LIN {X 0,Y 227.734,Z 309.956,A -85,B 0,C 180,E1 -22009.411,E2 -22009.411} C_VEL
LIN {X 0,Y 228.361,Z 312.963,A -85,B 0,C 180,E1 -22009.7,E2 -22009.7} C_VEL
LIN {X 0,Y 228.678,Z 315.581,A -85,B 0,C 180,E1 -22009.892,E2 -22009.892} C_VEL
LIN {X 0,Y 228.78,Z 319.404,A -85,B 0,C 180,E1 -22010.083,E2 -22010.083} C_VEL
LIN {X 0,Y 227.94,Z 325.239,A -85,B 0,C 180,E1 -22010.131,E2 -22010.131} C_VEL
LIN {X 0,Y 223.626,Z 340.721,A -85,B 0,C 180,E1 -22009.737,E2 -22009.737} C_VEL
LIN {X 0,Y 222.68,Z 346.699,A -85,B 0,C 180,E1 -22009.764,E2 -22009.764} C_VEL
LIN {X 0,Y 221.395,Z 364.438,A -85,B 0,C 180,E1 -22010.365,E2 -22010.365} C_VEL
LIN {X 0,Y 219.577,Z 377.351,A -85,B 0,C 180,E1 -22011.087,E2 -22011.087} C_VEL
LIN {X 0,Y 216.967,Z 389.201,A -85,B 0,C 180,E1 -22012.016,E2 -22012.016} C_VEL
LIN {X 0,Y 213.494,Z 401.606,A -85,B 0,C 180,E1 -22013.369,E2 -22013.369} C_VEL
LIN {X 0,Y 209.863,Z 412.686,A -85,B 0,C 180,E1 -22015.005,E2 -22015.005} C_VEL
LIN {X 0,Y 205.863,Z 422.69,A -85,B 0,C 180,E1 -22016.891,E2 -22016.891} C_VEL
LIN {X 0,Y 201.879,Z 431.756,A -85,B 0,C 180,E1 -22019.102,E2 -22019.102} C_VEL
LIN {X 0,Y 197.507,Z 440.623,A -85,B 0,C 180,E1 -22021.868,E2 -22021.868} C_VEL
LIN {X 0,Y 193.752,Z 447.781,A -85,B 0,C 180,E1 -22024.772,E2 -22024.772} C_VEL
LIN {X 0,Y 190.188,Z 454.335,A -85,B 0,C 180,E1 -22028.311,E2 -22028.311} C_VEL
LIN {X 0,Y 187.599,Z 458.703,A -85,B 0,C 180,E1 -22031.429,E2 -22031.429} C_VEL
LIN {X 0,Y 185.534,Z 462.024,A -85,B 0,C 180,E1 -22034.621,E2 -22034.621} C_VEL
LIN {X 0,Y 183.936,Z 464.98,A -85,B 0,C 180,E1 -22038.983,E2 -22038.983} C_VEL
LIN {X 0,Y 183.438,Z 465.859,A -85,B 0,C 180,E1 -22041.181,E2 -22041.181} C_VEL
LIN {X 0,Y 183.187,Z 466.397,A -85,B 0,C 180,E1 -22045.596,E2 -22045.596} C_VEL
LIN {X 0,Y 183.294,Z 466.092,A -85,B 0,C 180,E1 -22047.799,E2 -22047.799} C_VEL
LIN {X 0,Y 183.434,Z 465.393,A -85,B 0,C 180,E1 -22049.996,E2 -22049.996} C_VEL
LIN {X 0,Y 183.307,Z 464.225,A -85,B 0,C 180,E1 -22052.193,E2 -22052.193} C_VEL
LIN {X 0,Y 183.249,Z 461.69,A -85,B 0,C 180,E1 -22055.497,E2 -22055.497} C_VEL
LIN {X 0,Y 183.514,Z 458.117,A -85,B 0,C 180,E1 -22058.807,E2 -22058.807} C_VEL
LIN {X 0,Y 184.091,Z 453.401,A -85,B 0,C 180,E1 -22062.115,E2 -22062.115} C_VEL
LIN {X 0,Y 185.272,Z 447.418,A -85,B 0,C 180,E1 -22065.393,E2 -22065.393} C_VEL
LIN {X 0,Y 186.959,Z 439.943,A -85,B 0,C 180,E1 -22068.628,E2 -22068.628} C_VEL
LIN {X 0,Y 188.929,Z 431.416,A -85,B 0,C 180,E1 -22071.568,E2 -22071.568} C_VEL
LIN {X 0,Y 191.232,Z 422.023,A -85,B 0,C 180,E1 -22074.126,E2 -22074.126} C_VEL
LIN {X 0,Y 193.478,Z 411.462,A -85,B 0,C 180,E1 -22076.415,E2 -22076.415} C_VEL
LIN {X 0,Y 196.066,Z 399.786,A -85,B 0,C 180,E1 -22078.348,E2 -22078.348} C_VEL
LIN {X 0,Y 198.006,Z 388.456,A -85,B 0,C 180,E1 -22079.788,E2 -22079.788} C_VEL
LIN {X 0,Y 199.765,Z 374.91,A -85,B 0,C 180,E1 -22081.032,E2 -22081.032} C_VEL
LIN {X 0,Y 201.01,Z 362.184,A -85,B 0,C 180,E1 -22081.787,E2 -22081.787} C_VEL
LIN {X 0,Y 202.936,Z 313.059,A -85,B 0,C 180,E1 -22083.497,E2 -22083.497} C_VEL
LIN {X 0,Y 200.019,Z 283.806,A -85,B 0,C 180,E1 -22085.145,E2 -22085.145} C_VEL
LIN {X 0,Y 193.869,Z 267.805,A -85,B 0,C 180,E1 -22086.89,E2 -22086.89} C_VEL
LIN {X 0,Y 188.216,Z 255.397,A -85,B 0,C 180,E1 -22088.52,E2 -22088.52} C_VEL
LIN {X 0,Y 187.127,Z 252.759,A -85,B 0,C 180,E1 -22088.908,E2 -22088.908} C_VEL
LIN {X 0,Y 185.484,Z 246.381,A -85,B 0,C 180,E1 -22092.44,E2 -22092.44} C_VEL
LIN {X 0,Y 185.502,Z 246.379,A -85,B 0,C 180,E1 -22097.003,E2 -22097.003} C_VEL
LIN {X 0,Y 185.516,Z 246.376,A -85,B 0,C 180,E1 -22099.908,E2 -22099.908} C_VEL
LIN {X 0,Y 185.522,Z 246.375,A -85,B 0,C 180,E1 -22102.691,E2 -22102.691} C_VEL
LIN {X 0,Y 185.518,Z 246.378,A -85,B 0,C 180,E1 -22107.97,E2 -22107.97} C_VEL
LIN {X 0,Y 185.556,Z 246.37,A -85,B 0,C 180,E1 -22110.572,E2 -22110.572} C_VEL
LIN {X 0,Y 185.58,Z 246.37,A -85,B 0,C 180,E1 -22115.382,E2 -22115.382} C_VEL
LIN {X 0,Y 185.682,Z 246.353,A -85,B 0,C 180,E1 -22121.098,E2 -22121.098} C_VEL
LIN {X 0,Y 185.692,Z 246.346,A -85,B 0,C 180,E1 -22126.875,E2 -22126.875} C_VEL
LIN {X 0,Y 185.95,Z 246.318,A -85,B 0,C 180,E1 -22131.305,E2 -22131.305} C_VEL
LIN {X 0,Y 186.169,Z 246.288,A -85,B 0,C 180,E1 -22137.837,E2 -22137.837} C_VEL
LIN {X 0,Y 186.364,Z 246.247,A -85,B 0,C 180,E1 -22140,E2 -22140} C_VEL
LIN {X 0,Y 185.871,Z 246.312,A -85,B 0,C 180,E1 -22144.337,E2 -22144.337} C_VEL
LIN {X 0,Y 185.943,Z 246.323,A -85,B 0,C 180,E1 -22148.696,E2 -22148.696} C_VEL
LIN {X 0,Y 185.672,Z 246.328,A -85,B 0,C 180,E1 -22153.127,E2 -22153.127} C_VEL
LIN {X 0,Y 185.596,Z 246.362,A -85,B 0,C 180,E1 -22158.824,E2 -22158.824} C_VEL
LIN {X 0,Y 185.551,Z 246.368,A -85,B 0,C 180,E1 -22164.65,E2 -22164.65} C_VEL
LIN {X 0,Y 185.553,Z 246.366,A -85,B 0,C 180,E1 -22169.498,E2 -22169.498} C_VEL
LIN {X 0,Y 185.489,Z 246.374,A -85,B 0,C 180,E1 -22174.635,E2 -22174.635} C_VEL
LIN {X 0,Y 185.523,Z 246.374,A -85,B 0,C 180,E1 -22177.309,E2 -22177.309} C_VEL
LIN {X 0,Y 185.513,Z 246.375,A -85,B 0,C 180,E1 -22180.752,E2 -22180.752} C_VEL
LIN {X 0,Y 185.498,Z 246.365,A -85,B 0,C 180,E1 -22183.969,E2 -22183.969} C_VEL
LIN {X 0,Y 185.45,Z 246.381,A -85,B 0,C 180,E1 -22189.284,E2 -22189.284} C_VEL
LIN {X 0,Y 185.487,Z 246.363,A -85,B 0,C 180,E1 -22192.72,E2 -22192.72} C_VEL
LIN {X 0,Y 185.531,Z 246.374,A -85,B 0,C 180,E1 -22197.981,E2 -22197.981} C_VEL
LIN {X 0,Y 185.591,Z 246.368,A -85,B 0,C 180,E1 -22202.234,E2 -22202.234} C_VEL
LIN {X 0,Y 186.635,Z 249.244,A -85,B 0,C 180,E1 -22202.601,E2 -22202.601} C_VEL
LIN {X 0,Y 188.21,Z 251.839,A -85,B 0,C 180,E1 -22203.041,E2 -22203.041} C_VEL
LIN {X 0,Y 195.644,Z 265.32,A -85,B 0,C 180,E1 -22205.051,E2 -22205.051} C_VEL
LIN {X 0,Y 203.794,Z 282.946,A -85,B 0,C 180,E1 -22207.16,E2 -22207.16} C_VEL
LIN {X 0,Y 204.128,Z 284.701,A -85,B 0,C 180,E1 -22207.284,E2 -22207.284} C_VEL
LIN {X 0,Y 201.326,Z 346.607,A -85,B 0,C 180,E1 -22209.385,E2 -22209.385} C_VEL
LIN {X 0,Y 200.191,Z 359.424,A -85,B 0,C 180,E1 -22210.19,E2 -22210.19} C_VEL
LIN {X 0,Y 198.771,Z 371.41,A -85,B 0,C 180,E1 -22211.317,E2 -22211.317} C_VEL
LIN {X 0,Y 197.058,Z 383.513,A -85,B 0,C 180,E1 -22212.894,E2 -22212.894} C_VEL
LIN {X 0,Y 194.731,Z 395.058,A -85,B 0,C 180,E1 -22214.837,E2 -22214.837} C_VEL
LIN {X 0,Y 192.498,Z 405.426,A -85,B 0,C 180,E1 -22217.084,E2 -22217.084} C_VEL
LIN {X 0,Y 190.411,Z 413.923,A -85,B 0,C 180,E1 -22219.37,E2 -22219.37} C_VEL
LIN {X 0,Y 188.567,Z 421.735,A -85,B 0,C 180,E1 -22221.971,E2 -22221.971} C_VEL
LIN {X 0,Y 186.607,Z 429.386,A -85,B 0,C 180,E1 -22225.144,E2 -22225.144} C_VEL
LIN {X 0,Y 185.061,Z 436.428,A -85,B 0,C 180,E1 -22228.916,E2 -22228.916} C_VEL
LIN {X 0,Y 184.111,Z 441.123,A -85,B 0,C 180,E1 -22232.192,E2 -22232.192} C_VEL
LIN {X 0,Y 183.6,Z 444.798,A -85,B 0,C 180,E1 -22235.583,E2 -22235.583} C_VEL
LIN {X 0,Y 183.157,Z 447.315,A -85,B 0,C 180,E1 -22238.832,E2 -22238.832} C_VEL
LIN {X 0,Y 183.079,Z 448.541,A -85,B 0,C 180,E1 -22241.069,E2 -22241.069} C_VEL
LIN {X 0,Y 183.222,Z 449.315,A -85,B 0,C 180,E1 -22243.309,E2 -22243.309} C_VEL
LIN {X 0,Y 183.826,Z 449.725,A -85,B 0,C 180,E1 -22247.098,E2 -22247.098} C_VEL
LIN {X 0,Y 184.615,Z 449.269,A -85,B 0,C 180,E1 -22250.039,E2 -22250.039} C_VEL
LIN {X 0,Y 185.457,Z 448.402,A -85,B 0,C 180,E1 -22252.271,E2 -22252.271} C_VEL
LIN {X 0,Y 187.367,Z 446.14,A -85,B 0,C 180,E1 -22255.811,E2 -22255.811} C_VEL
LIN {X 0,Y 190.25,Z 441.994,A -85,B 0,C 180,E1 -22259.915,E2 -22259.915} C_VEL
LIN {X 0,Y 193.424,Z 436.987,A -85,B 0,C 180,E1 -22263.311,E2 -22263.311} C_VEL
LIN {X 0,Y 197.285,Z 430.362,A -85,B 0,C 180,E1 -22266.634,E2 -22266.634} C_VEL
LIN {X 0,Y 200.62,Z 424.064,A -85,B 0,C 180,E1 -22269.092,E2 -22269.092} C_VEL
LIN {X 0,Y 204.219,Z 416.437,A -85,B 0,C 180,E1 -22271.489,E2 -22271.489} C_VEL
LIN {X 0,Y 208.23,Z 407.146,A -85,B 0,C 180,E1 -22273.78,E2 -22273.78} C_VEL
LIN {X 0,Y 211.993,Z 396.993,A -85,B 0,C 180,E1 -22275.733,E2 -22275.733} C_VEL
LIN {X 0,Y 215.57,Z 385.061,A -85,B 0,C 180,E1 -22277.528,E2 -22277.528} C_VEL
LIN {X 0,Y 218.293,Z 373.848,A -85,B 0,C 180,E1 -22278.812,E2 -22278.812} C_VEL
LIN {X 0,Y 220.701,Z 361.29,A -85,B 0,C 180,E1 -22279.839,E2 -22279.839} C_VEL
LIN {X 0,Y 222.341,Z 348.203,A -85,B 0,C 180,E1 -22280.575,E2 -22280.575} C_VEL
LIN {X 0,Y 224.397,Z 317.273,A -85,B 0,C 180,E1 -22281.533,E2 -22281.533} C_VEL
LIN {X 0,Y 225.036,Z 305.015,A -85,B 0,C 180,E1 -22281.92,E2 -22281.92} C_VEL
LIN {X 0,Y 221.488,Z 297.767,A -85,B 0,C 180,E1 -22283.216,E2 -22283.216} C_VEL
LIN {X 0,Y 214.719,Z 286.12,A -85,B 0,C 180,E1 -22285.804,E2 -22285.804} C_VEL
LIN {X 0,Y 208.914,Z 277.344,A -85,B 0,C 180,E1 -22288.222,E2 -22288.222} C_VEL
LIN {X 0,Y 204.365,Z 270.883,A -85,B 0,C 180,E1 -22290.294,E2 -22290.294} C_VEL
LIN {X 0,Y 201.151,Z 266.565,A -85,B 0,C 180,E1 -22291.869,E2 -22291.869} C_VEL
LIN {X 0,Y 197.768,Z 262.05,A -85,B 0,C 180,E1 -22293.662,E2 -22293.662} C_VEL
LIN {X 0,Y 195.237,Z 259.03,A -85,B 0,C 180,E1 -22295.087,E2 -22295.087} C_VEL
LIN {X 0,Y 194.199,Z 257.394,A -85,B 0,C 180,E1 -22295.729,E2 -22295.729} C_VEL
LIN {X 0,Y 191.635,Z 254.934,A -85,B 0,C 180,E1 -22297.28,E2 -22297.28} C_VEL
LIN {X 0,Y 190.199,Z 252.182,A -85,B 0,C 180,E1 -22298.314,E2 -22298.314} C_VEL
LIN {X 0,Y 187.632,Z 250.55,A -85,B 0,C 180,E1 -22300.014,E2 -22300.014} C_VEL
LIN {X 0,Y 186.14,Z 248.277,A -85,B 0,C 180,E1 -22301.197,E2 -22301.197} C_VEL
LIN {X 0,Y 185.645,Z 246.353,A -85,B 0,C 180,E1 -22301.795,E2 -22301.795} C_VEL
LIN {X 0,Y 185.706,Z 246.354,A -85,B 0,C 180,E1 -22306.875,E2 -22306.875} C_VEL
LIN {X 0,Y 185.969,Z 246.321,A -85,B 0,C 180,E1 -22311.305,E2 -22311.305} C_VEL
LIN {X 0,Y 186.191,Z 246.278,A -85,B 0,C 180,E1 -22317.837,E2 -22317.837} C_VEL
LIN {X 0,Y 186.386,Z 246.263,A -85,B 0,C 180,E1 -22320,E2 -22320} C_VEL
LIN {X 0,Y 185.88,Z 246.322,A -85,B 0,C 180,E1 -22324.337,E2 -22324.337} C_VEL
LIN {X 0,Y 185.961,Z 246.308,A -85,B 0,C 180,E1 -22328.695,E2 -22328.695} C_VEL
LIN {X 0,Y 185.705,Z 246.339,A -85,B 0,C 180,E1 -22333.124,E2 -22333.124} C_VEL
LIN {X 0,Y 185.645,Z 246.347,A -85,B 0,C 180,E1 -22337.629,E2 -22337.629} C_VEL
LIN {X 0,Y 185.54,Z 246.362,A -85,B 0,C 180,E1 -22342.258,E2 -22342.258} C_VEL
LIN {X 0,Y 185.512,Z 246.377,A -85,B 0,C 180,E1 -22346.13,E2 -22346.13} C_VEL
LIN {X 0,Y 186.698,Z 249.68,A -85,B 0,C 180,E1 -22349.719,E2 -22349.719} C_VEL
LIN {X 0,Y 188.881,Z 253.094,A -85,B 0,C 180,E1 -22351.394,E2 -22351.394} C_VEL
LIN {X 0,Y 192.129,Z 257.04,A -85,B 0,C 180,E1 -22353.57,E2 -22353.57} C_VEL
LIN {X 0,Y 195.804,Z 262.28,A -85,B 0,C 180,E1 -22355.839,E2 -22355.839} C_VEL
LIN {X 0,Y 200.633,Z 269.693,A -85,B 0,C 180,E1 -22358.525,E2 -22358.525} C_VEL
LIN {X 0,Y 204.706,Z 276.314,A -85,B 0,C 180,E1 -22360.576,E2 -22360.576} C_VEL
LIN {X 0,Y 209.411,Z 284.218,A -85,B 0,C 180,E1 -22362.748,E2 -22362.748} C_VEL
LIN {X 0,Y 215.826,Z 296.589,A -85,B 0,C 180,E1 -22365.489,E2 -22365.489} C_VEL
LIN {X 0,Y 221.263,Z 308.869,A -85,B 0,C 180,E1 -22367.659,E2 -22367.659} C_VEL
LIN {X 0,Y 223.269,Z 314.09,A -85,B 0,C 180,E1 -22368.443,E2 -22368.443} C_VEL
LIN {X 0,Y 224.222,Z 322.363,A -85,B 0,C 180,E1 -22369.067,E2 -22369.067} C_VEL
LIN {X 0,Y 222.68,Z 346.699,A -85,B 0,C 180,E1 -22369.764,E2 -22369.764} C_VEL
LIN {X 0,Y 221.783,Z 352.547,A -85,B 0,C 180,E1 -22369.794,E2 -22369.794} C_VEL
LIN {X 0,Y 218.936,Z 362.031,A -85,B 0,C 180,E1 -22369.572,E2 -22369.572} C_VEL
LIN {X 0,Y 215.816,Z 371.411,A -85,B 0,C 180,E1 -22369.523,E2 -22369.523} C_VEL
LIN {X 0,Y 214.468,Z 377.081,A -85,B 0,C 180,E1 -22369.78,E2 -22369.78} C_VEL
LIN {X 0,Y 211.98,Z 388.215,A -85,B 0,C 180,E1 -22370.649,E2 -22370.649} C_VEL
LIN {X 0,Y 208.387,Z 400.753,A -85,B 0,C 180,E1 -22372.012,E2 -22372.012} C_VEL
LIN {X 0,Y 204.599,Z 411.931,A -85,B 0,C 180,E1 -22373.662,E2 -22373.662} C_VEL
LIN {X 0,Y 200.434,Z 422.037,A -85,B 0,C 180,E1 -22375.569,E2 -22375.569} C_VEL
LIN {X 0,Y 195.821,Z 431.971,A -85,B 0,C 180,E1 -22378.036,E2 -22378.036} C_VEL
LIN {X 0,Y 191.284,Z 440.747,A -85,B 0,C 180,E1 -22380.867,E2 -22380.867} C_VEL
LIN {X 0,Y 187.32,Z 447.797,A -85,B 0,C 180,E1 -22383.841,E2 -22383.841} C_VEL
LIN {X 0,Y 183.602,Z 454.272,A -85,B 0,C 180,E1 -22387.492,E2 -22387.492} C_VEL
LIN {X 0,Y 180.864,Z 458.577,A -85,B 0,C 180,E1 -22390.711,E2 -22390.711} C_VEL
LIN {X 0,Y 178.672,Z 461.84,A -85,B 0,C 180,E1 -22394.015,E2 -22394.015} C_VEL
LIN {X 0,Y 176.945,Z 464.742,A -85,B 0,C 180,E1 -22398.542,E2 -22398.542} C_VEL
LIN {X 0,Y 176.13,Z 466.002,A -85,B 0,C 180,E1 -22403.121,E2 -22403.121} C_VEL
LIN {X 0,Y 176.121,Z 466.025,A -85,B 0,C 180,E1 -22406.036,E2 -22406.036} C_VEL
LIN {X 0,Y 176.35,Z 464.984,A -85,B 0,C 180,E1 -22409.996,E2 -22409.996} C_VEL
LIN {X 0,Y 176.135,Z 462.585,A -85,B 0,C 180,E1 -22414.027,E2 -22414.027} C_VEL
LIN {X 0,Y 176.328,Z 458.879,A -85,B 0,C 180,E1 -22418.014,E2 -22418.014} C_VEL
LIN {X 0,Y 176.847,Z 454.496,A -85,B 0,C 180,E1 -22421.456,E2 -22421.456} C_VEL
LIN {X 0,Y 177.874,Z 448.896,A -85,B 0,C 180,E1 -22424.876,E2 -22424.876} C_VEL
LIN {X 0,Y 179.51,Z 441.896,A -85,B 0,C 180,E1 -22428.246,E2 -22428.246} C_VEL
LIN {X 0,Y 181.196,Z 434.913,A -85,B 0,C 180,E1 -22430.946,E2 -22430.946} C_VEL
LIN {X 0,Y 183.506,Z 426.06,A -85,B 0,C 180,E1 -22433.705,E2 -22433.705} C_VEL
LIN {X 0,Y 185.99,Z 415.328,A -85,B 0,C 180,E1 -22436.352,E2 -22436.352} C_VEL
LIN {X 0,Y 188.419,Z 404.701,A -85,B 0,C 180,E1 -22438.389,E2 -22438.389} C_VEL
LIN {X 0,Y 190.728,Z 392.883,A -85,B 0,C 180,E1 -22440.128,E2 -22440.128} C_VEL
LIN {X 0,Y 192.494,Z 381.883,A -85,B 0,C 180,E1 -22441.342,E2 -22441.342} C_VEL
LIN {X 0,Y 194.096,Z 368.944,A -85,B 0,C 180,E1 -22442.35,E2 -22442.35} C_VEL
LIN {X 0,Y 195.027,Z 355.86,A -85,B 0,C 180,E1 -22442.992,E2 -22442.992} C_VEL
LIN {X 0,Y 196.718,Z 313.925,A -85,B 0,C 180,E1 -22444.451,E2 -22444.451} C_VEL
LIN {X 0,Y 194.037,Z 285.989,A -85,B 0,C 180,E1 -22446.081,E2 -22446.081} C_VEL
LIN {X 0,Y 187.457,Z 268.879,A -85,B 0,C 180,E1 -22448.065,E2 -22448.065} C_VEL
LIN {X 0,Y 181.497,Z 256.082,A -85,B 0,C 180,E1 -22449.898,E2 -22449.898} C_VEL
LIN {X 0,Y 179.751,Z 252.309,A -85,B 0,C 180,E1 -22450.538,E2 -22450.538} C_VEL
LIN {X 0,Y 178.437,Z 247.259,A -85,B 0,C 180,E1 -22453.565,E2 -22453.565} C_VEL
LIN {X 0,Y 178.431,Z 247.261,A -85,B 0,C 180,E1 -22458.436,E2 -22458.436} C_VEL
LIN {X 0,Y 178.452,Z 247.258,A -85,B 0,C 180,E1 -22461.953,E2 -22461.953} C_VEL
LIN {X 0,Y 178.463,Z 247.253,A -85,B 0,C 180,E1 -22466.542,E2 -22466.542} C_VEL
LIN {X 0,Y 178.497,Z 247.249,A -85,B 0,C 180,E1 -22470.003,E2 -22470.003} C_VEL
LIN {X 0,Y 178.509,Z 247.249,A -85,B 0,C 180,E1 -22474.872,E2 -22474.872} C_VEL
LIN {X 0,Y 178.627,Z 247.233,A -85,B 0,C 180,E1 -22480.753,E2 -22480.753} C_VEL
LIN {X 0,Y 178.622,Z 247.227,A -85,B 0,C 180,E1 -22486.345,E2 -22486.345} C_VEL
LIN {X 0,Y 178.879,Z 247.201,A -85,B 0,C 180,E1 -22490.958,E2 -22490.958} C_VEL
LIN {X 0,Y 179.115,Z 247.167,A -85,B 0,C 180,E1 -22497.752,E2 -22497.752} C_VEL
LIN {X 0,Y 179.328,Z 247.121,A -85,B 0,C 180,E1 -22500,E2 -22500} C_VEL
LIN {X 0,Y 178.819,Z 247.191,A -85,B 0,C 180,E1 -22504.509,E2 -22504.509} C_VEL
LIN {X 0,Y 178.873,Z 247.201,A -85,B 0,C 180,E1 -22509.042,E2 -22509.042} C_VEL
LIN {X 0,Y 178.599,Z 247.203,A -85,B 0,C 180,E1 -22513.657,E2 -22513.657} C_VEL
LIN {X 0,Y 178.525,Z 247.245,A -85,B 0,C 180,E1 -22519.153,E2 -22519.153} C_VEL
LIN {X 0,Y 178.494,Z 247.251,A -85,B 0,C 180,E1 -22525.118,E2 -22525.118} C_VEL
LIN {X 0,Y 178.497,Z 247.246,A -85,B 0,C 180,E1 -22529.997,E2 -22529.997} C_VEL
LIN {X 0,Y 178.468,Z 247.248,A -85,B 0,C 180,E1 -22534.227,E2 -22534.227} C_VEL
LIN {X 0,Y 178.425,Z 247.251,A -85,B 0,C 180,E1 -22539.067,E2 -22539.067} C_VEL
LIN {X 0,Y 178.428,Z 247.258,A -85,B 0,C 180,E1 -22542.037,E2 -22542.037} C_VEL
LIN {X 0,Y 178.408,Z 247.239,A -85,B 0,C 180,E1 -22545.16,E2 -22545.16} C_VEL
LIN {X 0,Y 178.39,Z 247.257,A -85,B 0,C 180,E1 -22548.465,E2 -22548.465} C_VEL
LIN {X 0,Y 178.406,Z 247.247,A -85,B 0,C 180,E1 -22553.789,E2 -22553.789} C_VEL
LIN {X 0,Y 178.474,Z 247.252,A -85,B 0,C 180,E1 -22556.553,E2 -22556.553} C_VEL
LIN {X 0,Y 178.547,Z 247.245,A -85,B 0,C 180,E1 -22560.699,E2 -22560.699} C_VEL
LIN {X 0,Y 179.59,Z 250.168,A -85,B 0,C 180,E1 -22561.114,E2 -22561.114} C_VEL
LIN {X 0,Y 180.987,Z 252.16,A -85,B 0,C 180,E1 -22561.524,E2 -22561.524} C_VEL
LIN {X 0,Y 189.856,Z 268.184,A -85,B 0,C 180,E1 -22564.097,E2 -22564.097} C_VEL
LIN {X 0,Y 197.504,Z 284.764,A -85,B 0,C 180,E1 -22566.195,E2 -22566.195} C_VEL
LIN {X 0,Y 197.914,Z 285.964,A -85,B 0,C 180,E1 -22566.315,E2 -22566.315} C_VEL
LIN {X 0,Y 195.012,Z 346.91,A -85,B 0,C 180,E1 -22568.432,E2 -22568.432} C_VEL
LIN {X 0,Y 193.842,Z 360.203,A -85,B 0,C 180,E1 -22569.305,E2 -22569.305} C_VEL
LIN {X 0,Y 192.26,Z 372.636,A -85,B 0,C 180,E1 -22570.521,E2 -22570.521} C_VEL
LIN {X 0,Y 190.621,Z 383.686,A -85,B 0,C 180,E1 -22572.02,E2 -22572.02} C_VEL
LIN {X 0,Y 188.197,Z 395.26,A -85,B 0,C 180,E1 -22574.019,E2 -22574.019} C_VEL
LIN {X 0,Y 185.861,Z 405.648,A -85,B 0,C 180,E1 -22576.335,E2 -22576.335} C_VEL
LIN {X 0,Y 183.468,Z 415.02,A -85,B 0,C 180,E1 -22578.963,E2 -22578.963} C_VEL
LIN {X 0,Y 181.232,Z 424.036,A -85,B 0,C 180,E1 -22582.204,E2 -22582.204} C_VEL
LIN {X 0,Y 179.229,Z 431.337,A -85,B 0,C 180,E1 -22585.507,E2 -22585.507} C_VEL
LIN {X 0,Y 177.956,Z 437.164,A -85,B 0,C 180,E1 -22588.873,E2 -22588.873} C_VEL
LIN {X 0,Y 177.009,Z 441.769,A -85,B 0,C 180,E1 -22592.28,E2 -22592.28} C_VEL
LIN {X 0,Y 176.512,Z 445.073,A -85,B 0,C 180,E1 -22595.493,E2 -22595.493} C_VEL
LIN {X 0,Y 176.031,Z 447.814,A -85,B 0,C 180,E1 -22599.193,E2 -22599.193} C_VEL
LIN {X 0,Y 175.992,Z 448.971,A -85,B 0,C 180,E1 -22601.521,E2 -22601.521} C_VEL
LIN {X 0,Y 176.178,Z 449.703,A -85,B 0,C 180,E1 -22603.851,E2 -22603.851} C_VEL
LIN {X 0,Y 176.8,Z 450.06,A -85,B 0,C 180,E1 -22607.44,E2 -22607.44} C_VEL
LIN {X 0,Y 177.779,Z 449.511,A -85,B 0,C 180,E1 -22610.844,E2 -22610.844} C_VEL
LIN {X 0,Y 178.714,Z 448.607,A -85,B 0,C 180,E1 -22613.159,E2 -22613.159} C_VEL
LIN {X 0,Y 180.562,Z 446.555,A -85,B 0,C 180,E1 -22616.461,E2 -22616.461} C_VEL
LIN {X 0,Y 183.012,Z 443.295,A -85,B 0,C 180,E1 -22619.95,E2 -22619.95} C_VEL
LIN {X 0,Y 185.958,Z 439.062,A -85,B 0,C 180,E1 -22623.191,E2 -22623.191} C_VEL
LIN {X 0,Y 189.502,Z 433.477,A -85,B 0,C 180,E1 -22626.398,E2 -22626.398} C_VEL
LIN {X 0,Y 193.542,Z 426.508,A -85,B 0,C 180,E1 -22629.455,E2 -22629.455} C_VEL
LIN {X 0,Y 197.343,Z 419.12,A -85,B 0,C 180,E1 -22631.985,E2 -22631.985} C_VEL
LIN {X 0,Y 201.29,Z 410.575,A -85,B 0,C 180,E1 -22634.29,E2 -22634.29} C_VEL
LIN {X 0,Y 205.31,Z 400.664,A -85,B 0,C 180,E1 -22636.385,E2 -22636.385} C_VEL
LIN {X 0,Y 208.868,Z 390.28,A -85,B 0,C 180,E1 -22638.112,E2 -22638.112} C_VEL
LIN {X 0,Y 212.075,Z 378.475,A -85,B 0,C 180,E1 -22639.658,E2 -22639.658} C_VEL
LIN {X 0,Y 214.821,Z 366.123,A -85,B 0,C 180,E1 -22640.799,E2 -22640.799} C_VEL
LIN {X 0,Y 216.882,Z 352.716,A -85,B 0,C 180,E1 -22641.68,E2 -22641.68} C_VEL
LIN {X 0,Y 218.112,Z 339.15,A -85,B 0,C 180,E1 -22642.205,E2 -22642.205} C_VEL
LIN {X 0,Y 220.017,Z 307.56,A -85,B 0,C 180,E1 -22643.166,E2 -22643.166} C_VEL
LIN {X 0,Y 215.993,Z 299.738,A -85,B 0,C 180,E1 -22644.72,E2 -22644.72} C_VEL
LIN {X 0,Y 210.726,Z 290.635,A -85,B 0,C 180,E1 -22646.871,E2 -22646.871} C_VEL
LIN {X 0,Y 204.333,Z 280.768,A -85,B 0,C 180,E1 -22649.721,E2 -22649.721} C_VEL
LIN {X 0,Y 198.393,Z 272.472,A -85,B 0,C 180,E1 -22652.686,E2 -22652.686} C_VEL
LIN {X 0,Y 195.133,Z 268.073,A -85,B 0,C 180,E1 -22654.497,E2 -22654.497} C_VEL
LIN {X 0,Y 192.475,Z 264.61,A -85,B 0,C 180,E1 -22656.09,E2 -22656.09} C_VEL
LIN {X 0,Y 191.38,Z 263.34,A -85,B 0,C 180,E1 -22656.77,E2 -22656.77} C_VEL
LIN {X 0,Y 188.683,Z 260.056,A -85,B 0,C 180,E1 -22658.562,E2 -22658.562} C_VEL
LIN {X 0,Y 187.947,Z 258.675,A -85,B 0,C 180,E1 -22659.12,E2 -22659.12} C_VEL
LIN {X 0,Y 185.323,Z 256.586,A -85,B 0,C 180,E1 -22660.987,E2 -22660.987} C_VEL
LIN {X 0,Y 183.706,Z 253.71,A -85,B 0,C 180,E1 -22662.394,E2 -22662.394} C_VEL
LIN {X 0,Y 183.349,Z 253.077,A -85,B 0,C 180,E1 -22662.718,E2 -22662.718} C_VEL
LIN {X 0,Y 180.637,Z 251.376,A -85,B 0,C 180,E1 -22665.063,E2 -22665.063} C_VEL
LIN {X 0,Y 179.143,Z 249.101,A -85,B 0,C 180,E1 -22666.674,E2 -22666.674} C_VEL
LIN {X 0,Y 178.68,Z 247.224,A -85,B 0,C 180,E1 -22667.434,E2 -22667.434} C_VEL
LIN {X 0,Y 178.9,Z 247.199,A -85,B 0,C 180,E1 -22670.959,E2 -22670.959} C_VEL
LIN {X 0,Y 179.137,Z 247.157,A -85,B 0,C 180,E1 -22677.751,E2 -22677.751} C_VEL
LIN {X 0,Y 179.35,Z 247.138,A -85,B 0,C 180,E1 -22680,E2 -22680} C_VEL
LIN {X 0,Y 178.828,Z 247.201,A -85,B 0,C 180,E1 -22684.508,E2 -22684.508} C_VEL
LIN {X 0,Y 178.894,Z 247.191,A -85,B 0,C 180,E1 -22689.041,E2 -22689.041} C_VEL
LIN {X 0,Y 178.633,Z 247.223,A -85,B 0,C 180,E1 -22693.654,E2 -22693.654} C_VEL
LIN {X 0,Y 178.55,Z 247.244,A -85,B 0,C 180,E1 -22699.151,E2 -22699.151} C_VEL
LIN {X 0,Y 178.506,Z 247.444,A -85,B 0,C 180,E1 -22701.964,E2 -22701.964} C_VEL
LIN {X 0,Y 178.794,Z 248.635,A -85,B 0,C 180,E1 -22703.352,E2 -22703.352} C_VEL
LIN {X 0,Y 180.079,Z 250.916,A -85,B 0,C 180,E1 -22704.817,E2 -22704.817} C_VEL
LIN {X 0,Y 181.998,Z 253.165,A -85,B 0,C 180,E1 -22706.674,E2 -22706.674} C_VEL
LIN {X 0,Y 184.744,Z 256.233,A -85,B 0,C 180,E1 -22709.003,E2 -22709.003} C_VEL
LIN {X 0,Y 188.202,Z 261.196,A -85,B 0,C 180,E1 -22711.662,E2 -22711.662} C_VEL
LIN {X 0,Y 189.922,Z 263.422,A -85,B 0,C 180,E1 -22712.845,E2 -22712.845} C_VEL
LIN {X 0,Y 194.146,Z 269.73,A -85,B 0,C 180,E1 -22715.553,E2 -22715.553} C_VEL
LIN {X 0,Y 197.865,Z 275.651,A -85,B 0,C 180,E1 -22717.705,E2 -22717.705} C_VEL
LIN {X 0,Y 201.811,Z 282.231,A -85,B 0,C 180,E1 -22719.791,E2 -22719.791} C_VEL
LIN {X 0,Y 204.483,Z 286.865,A -85,B 0,C 180,E1 -22721.11,E2 -22721.11} C_VEL
LIN {X 0,Y 210.337,Z 297.94,A -85,B 0,C 180,E1 -22723.806,E2 -22723.806} C_VEL
LIN {X 0,Y 215.358,Z 309.064,A -85,B 0,C 180,E1 -22725.969,E2 -22725.969} C_VEL
LIN {X 0,Y 218.542,Z 317.131,A -85,B 0,C 180,E1 -22727.29,E2 -22727.29} C_VEL
LIN {X 0,Y 219.21,Z 323.617,A -85,B 0,C 180,E1 -22727.784,E2 -22727.784} C_VEL
LIN {X 0,Y 216.71,Z 360.92,A -85,B 0,C 180,E1 -22728.907,E2 -22728.907} C_VEL
LIN {X 0,Y 214.907,Z 374.531,A -85,B 0,C 180,E1 -22729.615,E2 -22729.615} C_VEL
LIN {X 0,Y 214.468,Z 377.081,A -85,B 0,C 180,E1 -22729.78,E2 -22729.78} C_VEL
LIN {X 0,Y 212.874,Z 382.686,A -85,B 0,C 180,E1 -22730.061,E2 -22730.061} C_VEL
LIN {X 0,Y 208.471,Z 391.574,A -85,B 0,C 180,E1 -22730.293,E2 -22730.293} C_VEL
LIN {X 0,Y 203.705,Z 400.152,A -85,B 0,C 180,E1 -22730.713,E2 -22730.713} C_VEL
LIN {X 0,Y 201.557,Z 405.214,A -85,B 0,C 180,E1 -22731.296,E2 -22731.296} C_VEL
LIN {X 0,Y 197.48,Z 415.968,A -85,B 0,C 180,E1 -22733.09,E2 -22733.09} C_VEL
LIN {X 0,Y 193.288,Z 425.279,A -85,B 0,C 180,E1 -22735.062,E2 -22735.062} C_VEL
LIN {X 0,Y 189.06,Z 433.788,A -85,B 0,C 180,E1 -22737.382,E2 -22737.382} C_VEL
LIN {X 0,Y 184.36,Z 442.095,A -85,B 0,C 180,E1 -22740.291,E2 -22740.291} C_VEL
LIN {X 0,Y 180.35,Z 448.815,A -85,B 0,C 180,E1 -22743.374,E2 -22743.374} C_VEL
LIN {X 0,Y 177.053,Z 454.213,A -85,B 0,C 180,E1 -22746.611,E2 -22746.611} C_VEL
LIN {X 0,Y 174.16,Z 458.456,A -85,B 0,C 180,E1 -22749.937,E2 -22749.937} C_VEL
LIN {X 0,Y 171.838,Z 461.66,A -85,B 0,C 180,E1 -22753.361,E2 -22753.361} C_VEL
LIN {X 0,Y 169.972,Z 464.495,A -85,B 0,C 180,E1 -22758.065,E2 -22758.065} C_VEL
LIN {X 0,Y 169.08,Z 465.687,A -85,B 0,C 180,E1 -22762.833,E2 -22762.833} C_VEL
LIN {X 0,Y 169.036,Z 465.607,A -85,B 0,C 180,E1 -22766.242,E2 -22766.242} C_VEL
LIN {X 0,Y 169.267,Z 464.566,A -85,B 0,C 180,E1 -22769.996,E2 -22769.996} C_VEL
LIN {X 0,Y 169.046,Z 462.404,A -85,B 0,C 180,E1 -22773.809,E2 -22773.809} C_VEL
LIN {X 0,Y 169.162,Z 459.6,A -85,B 0,C 180,E1 -22777.155,E2 -22777.155} C_VEL
LIN {X 0,Y 169.618,Z 455.537,A -85,B 0,C 180,E1 -22780.74,E2 -22780.74} C_VEL
LIN {X 0,Y 170.729,Z 449.258,A -85,B 0,C 180,E1 -22784.903,E2 -22784.903} C_VEL
LIN {X 0,Y 172.432,Z 442.418,A -85,B 0,C 180,E1 -22788.407,E2 -22788.407} C_VEL
LIN {X 0,Y 174.19,Z 435.42,A -85,B 0,C 180,E1 -22791.285,E2 -22791.285} C_VEL
LIN {X 0,Y 176.473,Z 426.997,A -85,B 0,C 180,E1 -22794.085,E2 -22794.085} C_VEL
LIN {X 0,Y 179.073,Z 416.605,A -85,B 0,C 180,E1 -22796.822,E2 -22796.822} C_VEL
LIN {X 0,Y 181.182,Z 407.746,A -85,B 0,C 180,E1 -22798.679,E2 -22798.679} C_VEL
LIN {X 0,Y 183.574,Z 396.847,A -85,B 0,C 180,E1 -22800.474,E2 -22800.474} C_VEL
LIN {X 0,Y 185.74,Z 384.813,A -85,B 0,C 180,E1 -22801.979,E2 -22801.979} C_VEL
LIN {X 0,Y 187.403,Z 372.534,A -85,B 0,C 180,E1 -22803.093,E2 -22803.093} C_VEL
LIN {X 0,Y 188.578,Z 360.103,A -85,B 0,C 180,E1 -22803.819,E2 -22803.819} C_VEL
LIN {X 0,Y 190.534,Z 314.714,A -85,B 0,C 180,E1 -22805.47,E2 -22805.47} C_VEL
LIN {X 0,Y 188.042,Z 287.984,A -85,B 0,C 180,E1 -22807.096,E2 -22807.096} C_VEL
LIN {X 0,Y 181.882,Z 272.002,A -85,B 0,C 180,E1 -22809.065,E2 -22809.065} C_VEL
LIN {X 0,Y 176.211,Z 259.68,A -85,B 0,C 180,E1 -22810.923,E2 -22810.923} C_VEL
LIN {X 0,Y 173.78,Z 255.18,A -85,B 0,C 180,E1 -22811.731,E2 -22811.731} C_VEL
LIN {X 0,Y 172.347,Z 251.959,A -85,B 0,C 180,E1 -22812.295,E2 -22812.295} C_VEL
LIN {X 0,Y 171.371,Z 248.138,A -85,B 0,C 180,E1 -22814.658,E2 -22814.658} C_VEL
LIN {X 0,Y 171.358,Z 248.142,A -85,B 0,C 180,E1 -22818.988,E2 -22818.988} C_VEL
LIN {X 0,Y 171.4,Z 248.136,A -85,B 0,C 180,E1 -22822.044,E2 -22822.044} C_VEL
LIN {X 0,Y 171.384,Z 248.139,A -85,B 0,C 180,E1 -22825.084,E2 -22825.084} C_VEL
LIN {X 0,Y 171.424,Z 248.131,A -85,B 0,C 180,E1 -22830.53,E2 -22830.53} C_VEL
LIN {X 0,Y 171.441,Z 248.129,A -85,B 0,C 180,E1 -22835.799,E2 -22835.799} C_VEL
LIN {X 0,Y 171.582,Z 248.11,A -85,B 0,C 180,E1 -22840.872,E2 -22840.872} C_VEL
LIN {X 0,Y 171.543,Z 248.11,A -85,B 0,C 180,E1 -22845.77,E2 -22845.77} C_VEL
LIN {X 0,Y 171.817,Z 248.082,A -85,B 0,C 180,E1 -22850.583,E2 -22850.583} C_VEL
LIN {X 0,Y 171.778,Z 248.087,A -85,B 0,C 180,E1 -22855.307,E2 -22855.307} C_VEL
LIN {X 0,Y 172.291,Z 247.996,A -85,B 0,C 180,E1 -22860,E2 -22860} C_VEL
LIN {X 0,Y 171.767,Z 248.07,A -85,B 0,C 180,E1 -22864.694,E2 -22864.694} C_VEL
LIN {X 0,Y 171.812,Z 248.079,A -85,B 0,C 180,E1 -22869.417,E2 -22869.417} C_VEL
LIN {X 0,Y 171.514,Z 248.082,A -85,B 0,C 180,E1 -22874.233,E2 -22874.233} C_VEL
LIN {X 0,Y 171.45,Z 248.127,A -85,B 0,C 180,E1 -22879.501,E2 -22879.501} C_VEL
LIN {X 0,Y 171.432,Z 248.13,A -85,B 0,C 180,E1 -22885.612,E2 -22885.612} C_VEL
LIN {X 0,Y 171.415,Z 248.131,A -85,B 0,C 180,E1 -22890.59,E2 -22890.59} C_VEL
LIN {X 0,Y 171.38,Z 248.132,A -85,B 0,C 180,E1 -22895.038,E2 -22895.038} C_VEL
LIN {X 0,Y 171.382,Z 248.129,A -85,B 0,C 180,E1 -22898.831,E2 -22898.831} C_VEL
LIN {X 0,Y 171.336,Z 248.125,A -85,B 0,C 180,E1 -22904.213,E2 -22904.213} C_VEL
LIN {X 0,Y 171.321,Z 248.141,A -85,B 0,C 180,E1 -22908.988,E2 -22908.988} C_VEL
LIN {X 0,Y 171.347,Z 248.125,A -85,B 0,C 180,E1 -22912.04,E2 -22912.04} C_VEL
LIN {X 0,Y 171.386,Z 248.132,A -85,B 0,C 180,E1 -22915.099,E2 -22915.099} C_VEL
LIN {X 0,Y 171.449,Z 248.229,A -85,B 0,C 180,E1 -22919.055,E2 -22919.055} C_VEL
LIN {X 0,Y 172.422,Z 250.96,A -85,B 0,C 180,E1 -22919.443,E2 -22919.443} C_VEL
LIN {X 0,Y 174.114,Z 253.336,A -85,B 0,C 180,E1 -22919.983,E2 -22919.983} C_VEL
LIN {X 0,Y 180.785,Z 264.868,A -85,B 0,C 180,E1 -22922.085,E2 -22922.085} C_VEL
LIN {X 0,Y 187.043,Z 277.089,A -85,B 0,C 180,E1 -22923.947,E2 -22923.947} C_VEL
LIN {X 0,Y 191.659,Z 287.476,A -85,B 0,C 180,E1 -22925.28,E2 -22925.28} C_VEL
LIN {X 0,Y 188.793,Z 347.071,A -85,B 0,C 180,E1 -22927.418,E2 -22927.418} C_VEL
LIN {X 0,Y 187.583,Z 360.193,A -85,B 0,C 180,E1 -22928.292,E2 -22928.292} C_VEL
LIN {X 0,Y 185.946,Z 372.714,A -85,B 0,C 180,E1 -22929.543,E2 -22929.543} C_VEL
LIN {X 0,Y 184.231,Z 383.832,A -85,B 0,C 180,E1 -22931.086,E2 -22931.086} C_VEL
LIN {X 0,Y 181.704,Z 395.44,A -85,B 0,C 180,E1 -22933.143,E2 -22933.143} C_VEL
LIN {X 0,Y 179.258,Z 405.854,A -85,B 0,C 180,E1 -22935.532,E2 -22935.532} C_VEL
LIN {X 0,Y 176.961,Z 414.392,A -85,B 0,C 180,E1 -22937.971,E2 -22937.971} C_VEL
LIN {X 0,Y 174.944,Z 422.236,A -85,B 0,C 180,E1 -22940.758,E2 -22940.758} C_VEL
LIN {X 0,Y 172.774,Z 429.925,A -85,B 0,C 180,E1 -22944.168,E2 -22944.168} C_VEL
LIN {X 0,Y 171.235,Z 436.086,A -85,B 0,C 180,E1 -22947.652,E2 -22947.652} C_VEL
LIN {X 0,Y 170.126,Z 440.99,A -85,B 0,C 180,E1 -22951.188,E2 -22951.188} C_VEL
LIN {X 0,Y 169.51,Z 444.774,A -85,B 0,C 180,E1 -22954.761,E2 -22954.761} C_VEL
LIN {X 0,Y 169.121,Z 446.748,A -85,B 0,C 180,E1 -22957.165,E2 -22957.165} C_VEL
LIN {X 0,Y 168.931,Z 448.3,A -85,B 0,C 180,E1 -22959.583,E2 -22959.583} C_VEL
LIN {X 0,Y 169.161,Z 450.09,A -85,B 0,C 180,E1 -22964.438,E2 -22964.438} C_VEL
LIN {X 0,Y 169.781,Z 450.396,A -85,B 0,C 180,E1 -22967.808,E2 -22967.808} C_VEL
LIN {X 0,Y 170.958,Z 449.756,A -85,B 0,C 180,E1 -22971.717,E2 -22971.717} C_VEL
LIN {X 0,Y 172.032,Z 448.814,A -85,B 0,C 180,E1 -22974.115,E2 -22974.115} C_VEL
LIN {X 0,Y 173.792,Z 446.967,A -85,B 0,C 180,E1 -22977.168,E2 -22977.168} C_VEL
LIN {X 0,Y 176.715,Z 443.348,A -85,B 0,C 180,E1 -22981.134,E2 -22981.134} C_VEL
LIN {X 0,Y 179.718,Z 439.254,A -85,B 0,C 180,E1 -22984.315,E2 -22984.315} C_VEL
LIN {X 0,Y 183.646,Z 433.352,A -85,B 0,C 180,E1 -22987.757,E2 -22987.757} C_VEL
LIN {X 0,Y 187.942,Z 426.254,A -85,B 0,C 180,E1 -22990.875,E2 -22990.875} C_VEL
LIN {X 0,Y 192.664,Z 417.279,A -85,B 0,C 180,E1 -22993.875,E2 -22993.875} C_VEL
LIN {X 0,Y 197.037,Z 408.027,A -85,B 0,C 180,E1 -22996.243,E2 -22996.243} C_VEL
LIN {X 0,Y 201.12,Z 397.942,A -85,B 0,C 180,E1 -22998.252,E2 -22998.252} C_VEL
LIN {X 0,Y 204.997,Z 386.08,A -85,B 0,C 180,E1 -23000.093,E2 -23000.093} C_VEL
LIN {X 0,Y 207.945,Z 374.964,A -85,B 0,C 180,E1 -23001.403,E2 -23001.403} C_VEL
LIN {X 0,Y 210.552,Z 362.663,A -85,B 0,C 180,E1 -23002.442,E2 -23002.442} C_VEL
LIN {X 0,Y 212.358,Z 349.702,A -85,B 0,C 180,E1 -23003.198,E2 -23003.198} C_VEL
LIN {X 0,Y 214.035,Z 327.85,A -85,B 0,C 180,E1 -23003.912,E2 -23003.912} C_VEL
LIN {X 0,Y 215.055,Z 310.041,A -85,B 0,C 180,E1 -23004.491,E2 -23004.491} C_VEL
LIN {X 0,Y 208.542,Z 298.049,A -85,B 0,C 180,E1 -23007.213,E2 -23007.213} C_VEL
LIN {X 0,Y 202.971,Z 289.041,A -85,B 0,C 180,E1 -23009.757,E2 -23009.757} C_VEL
LIN {X 0,Y 198.058,Z 281.813,A -85,B 0,C 180,E1 -23012.225,E2 -23012.225} C_VEL
LIN {X 0,Y 195.301,Z 277.889,A -85,B 0,C 180,E1 -23013.736,E2 -23013.736} C_VEL
LIN {X 0,Y 192.58,Z 274.128,A -85,B 0,C 180,E1 -23015.333,E2 -23015.333} C_VEL
LIN {X 0,Y 189.208,Z 269.702,A -85,B 0,C 180,E1 -23017.477,E2 -23017.477} C_VEL
LIN {X 0,Y 186.392,Z 266.139,A -85,B 0,C 180,E1 -23019.443,E2 -23019.443} C_VEL
LIN {X 0,Y 185.559,Z 265.034,A -85,B 0,C 180,E1 -23020.07,E2 -23020.07} C_VEL
LIN {X 0,Y 183.02,Z 262.482,A -85,B 0,C 180,E1 -23022.037,E2 -23022.037} C_VEL
LIN {X 0,Y 181.538,Z 259.804,A -85,B 0,C 180,E1 -23023.41,E2 -23023.41} C_VEL
LIN {X 0,Y 178.816,Z 257.758,A -85,B 0,C 180,E1 -23025.925,E2 -23025.925} C_VEL
LIN {X 0,Y 177.252,Z 255.039,A -85,B 0,C 180,E1 -23027.767,E2 -23027.767} C_VEL
LIN {X 0,Y 176.908,Z 254.074,A -85,B 0,C 180,E1 -23028.252,E2 -23028.252} C_VEL
LIN {X 0,Y 173.717,Z 252.08,A -85,B 0,C 180,E1 -23032.444,E2 -23032.444} C_VEL
LIN {X 0,Y 172.188,Z 249.592,A -85,B 0,C 180,E1 -23035.464,E2 -23035.464} C_VEL
LIN {X 0,Y 171.911,Z 248.067,A -85,B 0,C 180,E1 -23036.484,E2 -23036.484} C_VEL
LIN {X 0,Y 172.314,Z 248.014,A -85,B 0,C 180,E1 -23040,E2 -23040} C_VEL
LIN {X 0,Y 171.847,Z 248.064,A -85,B 0,C 180,E1 -23047.047,E2 -23047.047} C_VEL
LIN {X 0,Y 171.762,Z 248.081,A -85,B 0,C 180,E1 -23050.891,E2 -23050.891} C_VEL
LIN {X 0,Y 171.592,Z 248.115,A -85,B 0,C 180,E1 -23053.32,E2 -23053.32} C_VEL
LIN {X 0,Y 172.172,Z 250.287,A -85,B 0,C 180,E1 -23055.083,E2 -23055.083} C_VEL
LIN {X 0,Y 174.362,Z 252.97,A -85,B 0,C 180,E1 -23059.016,E2 -23059.016} C_VEL
LIN {X 0,Y 176.618,Z 254.409,A -85,B 0,C 180,E1 -23061.904,E2 -23061.904} C_VEL
LIN {X 0,Y 177.497,Z 255.944,A -85,B 0,C 180,E1 -23063.017,E2 -23063.017} C_VEL
LIN {X 0,Y 182.704,Z 262.533,A -85,B 0,C 180,E1 -23068.158,E2 -23068.158} C_VEL
LIN {X 0,Y 186.796,Z 268.333,A -85,B 0,C 180,E1 -23071.409,E2 -23071.409} C_VEL
LIN {X 0,Y 191.656,Z 275.867,A -85,B 0,C 180,E1 -23074.737,E2 -23074.737} C_VEL
LIN {X 0,Y 195.062,Z 281.415,A -85,B 0,C 180,E1 -23076.811,E2 -23076.811} C_VEL
LIN {X 0,Y 200.232,Z 290.288,A -85,B 0,C 180,E1 -23079.645,E2 -23079.645} C_VEL
LIN {X 0,Y 205.407,Z 300.357,A -85,B 0,C 180,E1 -23082.226,E2 -23082.226} C_VEL
LIN {X 0,Y 210.059,Z 310.402,A -85,B 0,C 180,E1 -23084.374,E2 -23084.374} C_VEL
LIN {X 0,Y 213.892,Z 320.154,A -85,B 0,C 180,E1 -23086.08,E2 -23086.08} C_VEL
LIN {X 0,Y 214.31,Z 324.72,A -85,B 0,C 180,E1 -23086.432,E2 -23086.432} C_VEL
LIN {X 0,Y 211.751,Z 361.175,A -85,B 0,C 180,E1 -23087.552,E2 -23087.552} C_VEL
LIN {X 0,Y 209.862,Z 374.715,A -85,B 0,C 180,E1 -23088.273,E2 -23088.273} C_VEL
LIN {X 0,Y 207.127,Z 387.19,A -85,B 0,C 180,E1 -23089.219,E2 -23089.219} C_VEL
LIN {X 0,Y 203.948,Z 398.322,A -85,B 0,C 180,E1 -23090.394,E2 -23090.394} C_VEL
LIN {X 0,Y 201.557,Z 405.214,A -85,B 0,C 180,E1 -23091.296,E2 -23091.296} C_VEL
LIN {X 0,Y 199.338,Z 410.186,A -85,B 0,C 180,E1 -23091.958,E2 -23091.958} C_VEL
LIN {X 0,Y 193.989,Z 417.989,A -85,B 0,C 180,E1 -23092.824,E2 -23092.824} C_VEL
LIN {X 0,Y 188.274,Z 425.3,A -85,B 0,C 180,E1 -23093.88,E2 -23093.88} C_VEL
LIN {X 0,Y 185.528,Z 429.469,A -85,B 0,C 180,E1 -23094.848,E2 -23094.848} C_VEL
LIN {X 0,Y 180.636,Z 438.284,A -85,B 0,C 180,E1 -23097.657,E2 -23097.657} C_VEL
LIN {X 0,Y 176.022,Z 445.679,A -85,B 0,C 180,E1 -23100.717,E2 -23100.717} C_VEL
LIN {X 0,Y 171.763,Z 452.281,A -85,B 0,C 180,E1 -23104.365,E2 -23104.365} C_VEL
LIN {X 0,Y 168.379,Z 457.076,A -85,B 0,C 180,E1 -23107.933,E2 -23107.933} C_VEL
LIN {X 0,Y 166.611,Z 459.49,A -85,B 0,C 180,E1 -23110.275,E2 -23110.275} C_VEL
LIN {X 0,Y 163.826,Z 463.07,A -85,B 0,C 180,E1 -23115.081,E2 -23115.081} C_VEL
LIN {X 0,Y 162.983,Z 464.235,A -85,B 0,C 180,E1 -23117.545,E2 -23117.545} C_VEL
LIN {X 0,Y 162.006,Z 465.371,A -85,B 0,C 180,E1 -23122.518,E2 -23122.518} C_VEL
LIN {X 0,Y 161.966,Z 465.186,A -85,B 0,C 180,E1 -23126.388,E2 -23126.388} C_VEL
LIN {X 0,Y 162.185,Z 464.147,A -85,B 0,C 180,E1 -23129.995,E2 -23129.995} C_VEL
LIN {X 0,Y 161.959,Z 462.219,A -85,B 0,C 180,E1 -23133.572,E2 -23133.572} C_VEL
LIN {X 0,Y 162.113,Z 459.071,A -85,B 0,C 180,E1 -23137.467,E2 -23137.467} C_VEL
LIN {X 0,Y 162.582,Z 454.941,A -85,B 0,C 180,E1 -23141.211,E2 -23141.211} C_VEL
LIN {X 0,Y 163.842,Z 448.591,A -85,B 0,C 180,E1 -23145.544,E2 -23145.544} C_VEL
LIN {X 0,Y 165.617,Z 441.669,A -85,B 0,C 180,E1 -23149.194,E2 -23149.194} C_VEL
LIN {X 0,Y 167.475,Z 434.581,A -85,B 0,C 180,E1 -23152.183,E2 -23152.183} C_VEL
LIN {X 0,Y 169.976,Z 426.061,A -85,B 0,C 180,E1 -23155.068,E2 -23155.068} C_VEL
LIN {X 0,Y 172.67,Z 415.474,A -85,B 0,C 180,E1 -23157.901,E2 -23157.901} C_VEL
LIN {X 0,Y 175.288,Z 405.015,A -85,B 0,C 180,E1 -23160.069,E2 -23160.069} C_VEL
LIN {X 0,Y 177.779,Z 393.531,A -85,B 0,C 180,E1 -23161.912,E2 -23161.912} C_VEL
LIN {X 0,Y 179.873,Z 381.677,A -85,B 0,C 180,E1 -23163.321,E2 -23163.321} C_VEL
LIN {X 0,Y 181.576,Z 368.904,A -85,B 0,C 180,E1 -23164.384,E2 -23164.384} C_VEL
LIN {X 0,Y 182.627,Z 355.692,A -85,B 0,C 180,E1 -23165.079,E2 -23165.079} C_VEL
LIN {X 0,Y 184.43,Z 315.595,A -85,B 0,C 180,E1 -23166.548,E2 -23166.548} C_VEL
LIN {X 0,Y 182.252,Z 290.559,A -85,B 0,C 180,E1 -23168.122,E2 -23168.122} C_VEL
LIN {X 0,Y 176.675,Z 275.761,A -85,B 0,C 180,E1 -23170.026,E2 -23170.026} C_VEL
LIN {X 0,Y 170.91,Z 263.116,A -85,B 0,C 180,E1 -23172.034,E2 -23172.034} C_VEL
LIN {X 0,Y 166.328,Z 254.462,A -85,B 0,C 180,E1 -23173.694,E2 -23173.694} C_VEL
LIN {X 0,Y 164.964,Z 251.59,A -85,B 0,C 180,E1 -23174.254,E2 -23174.254} C_VEL
LIN {X 0,Y 164.302,Z 249.019,A -85,B 0,C 180,E1 -23175.967,E2 -23175.967} C_VEL
LIN {X 0,Y 164.3,Z 249.018,A -85,B 0,C 180,E1 -23180.336,E2 -23180.336} C_VEL
LIN {X 0,Y 164.319,Z 249.019,A -85,B 0,C 180,E1 -23184.339,E2 -23184.339} C_VEL
LIN {X 0,Y 164.365,Z 249.01,A -85,B 0,C 180,E1 -23189.129,E2 -23189.129} C_VEL
LIN {X 0,Y 164.392,Z 249.007,A -85,B 0,C 180,E1 -23194.69,E2 -23194.69} C_VEL
LIN {X 0,Y 164.494,Z 248.994,A -85,B 0,C 180,E1 -23200.014,E2 -23200.014} C_VEL
LIN {X 0,Y 164.477,Z 248.994,A -85,B 0,C 180,E1 -23205.145,E2 -23205.145} C_VEL
LIN {X 0,Y 164.737,Z 248.963,A -85,B 0,C 180,E1 -23210.175,E2 -23210.175} C_VEL
LIN {X 0,Y 164.798,Z 248.947,A -85,B 0,C 180,E1 -23212.65,E2 -23212.65} C_VEL
LIN {X 0,Y 165.012,Z 248.924,A -85,B 0,C 180,E1 -23217.559,E2 -23217.559} C_VEL
LIN {X 0,Y 165.254,Z 248.87,A -85,B 0,C 180,E1 -23220,E2 -23220} C_VEL
LIN {X 0,Y 164.792,Z 248.956,A -85,B 0,C 180,E1 -23227.351,E2 -23227.351} C_VEL
LIN {X 0,Y 164.672,Z 248.959,A -85,B 0,C 180,E1 -23231.057,E2 -23231.057} C_VEL
LIN {X 0,Y 164.399,Z 248.99,A -85,B 0,C 180,E1 -23237.413,E2 -23237.413} C_VEL
LIN {X 0,Y 164.393,Z 249.006,A -85,B 0,C 180,E1 -23240,E2 -23240} C_VEL
LIN {X 0,Y 164.359,Z 249.012,A -85,B 0,C 180,E1 -23246.131,E2 -23246.131} C_VEL
LIN {X 0,Y 164.35,Z 249.013,A -85,B 0,C 180,E1 -23251.231,E2 -23251.231} C_VEL
LIN {X 0,Y 164.295,Z 249.019,A -85,B 0,C 180,E1 -23256.79,E2 -23256.79} C_VEL
LIN {X 0,Y 164.297,Z 249.011,A -85,B 0,C 180,E1 -23259.915,E2 -23259.915} C_VEL
LIN {X 0,Y 164.29,Z 249.01,A -85,B 0,C 180,E1 -23263.358,E2 -23263.358} C_VEL
LIN {X 0,Y 164.277,Z 248.998,A -85,B 0,C 180,E1 -23266.815,E2 -23266.815} C_VEL
LIN {X 0,Y 164.276,Z 249.017,A -85,B 0,C 180,E1 -23270.361,E2 -23270.361} C_VEL
LIN {X 0,Y 164.315,Z 249.017,A -85,B 0,C 180,E1 -23276.228,E2 -23276.228} C_VEL
LIN {X 0,Y 164.346,Z 249.01,A -85,B 0,C 180,E1 -23277.136,E2 -23277.136} C_VEL
LIN {X 0,Y 165.336,Z 251.794,A -85,B 0,C 180,E1 -23277.611,E2 -23277.611} C_VEL
LIN {X 0,Y 167.162,Z 254.308,A -85,B 0,C 180,E1 -23278.249,E2 -23278.249} C_VEL
LIN {X 0,Y 174.049,Z 265.767,A -85,B 0,C 180,E1 -23280.595,E2 -23280.595} C_VEL
LIN {X 0,Y 180.806,Z 278.803,A -85,B 0,C 180,E1 -23282.75,E2 -23282.75} C_VEL
LIN {X 0,Y 185.54,Z 289.431,A -85,B 0,C 180,E1 -23284.209,E2 -23284.209} C_VEL
LIN {X 0,Y 182.623,Z 347.445,A -85,B 0,C 180,E1 -23286.347,E2 -23286.347} C_VEL
LIN {X 0,Y 181.351,Z 360.2,A -85,B 0,C 180,E1 -23287.206,E2 -23287.206} C_VEL
LIN {X 0,Y 179.866,Z 371.659,A -85,B 0,C 180,E1 -23288.368,E2 -23288.368} C_VEL
LIN {X 0,Y 177.894,Z 383.974,A -85,B 0,C 180,E1 -23290.084,E2 -23290.084} C_VEL
LIN {X 0,Y 175.257,Z 395.617,A -85,B 0,C 180,E1 -23292.202,E2 -23292.202} C_VEL
LIN {X 0,Y 172.693,Z 406.057,A -85,B 0,C 180,E1 -23294.667,E2 -23294.667} C_VEL
LIN {X 0,Y 170.057,Z 415.487,A -85,B 0,C 180,E1 -23297.475,E2 -23297.475} C_VEL
LIN {X 0,Y 167.577,Z 424.537,A -85,B 0,C 180,E1 -23300.957,E2 -23300.957} C_VEL
LIN {X 0,Y 165.379,Z 431.866,A -85,B 0,C 180,E1 -23304.518,E2 -23304.518} C_VEL
LIN {X 0,Y 163.746,Z 438.557,A -85,B 0,C 180,E1 -23308.775,E2 -23308.775} C_VEL
LIN {X 0,Y 162.805,Z 442.989,A -85,B 0,C 180,E1 -23312.479,E2 -23312.479} C_VEL
LIN {X 0,Y 162.33,Z 445.596,A -85,B 0,C 180,E1 -23315.265,E2 -23315.265} C_VEL
LIN {X 0,Y 161.82,Z 448.762,A -85,B 0,C 180,E1 -23320.008,E2 -23320.008} C_VEL
LIN {X 0,Y 162.166,Z 450.476,A -85,B 0,C 180,E1 -23325.075,E2 -23325.075} C_VEL
LIN {X 0,Y 162.788,Z 450.729,A -85,B 0,C 180,E1 -23328.23,E2 -23328.23} C_VEL
LIN {X 0,Y 164.207,Z 449.999,A -85,B 0,C 180,E1 -23332.659,E2 -23332.659} C_VEL
LIN {X 0,Y 165.382,Z 449.022,A -85,B 0,C 180,E1 -23335.15,E2 -23335.15} C_VEL
LIN {X 0,Y 167.056,Z 447.376,A -85,B 0,C 180,E1 -23337.936,E2 -23337.936} C_VEL
LIN {X 0,Y 170.49,Z 443.4,A -85,B 0,C 180,E1 -23342.406,E2 -23342.406} C_VEL
LIN {X 0,Y 174.342,Z 438.36,A -85,B 0,C 180,E1 -23346.27,E2 -23346.27} C_VEL
LIN {X 0,Y 178.629,Z 432.105,A -85,B 0,C 180,E1 -23349.743,E2 -23349.743} C_VEL
LIN {X 0,Y 183.282,Z 424.593,A -85,B 0,C 180,E1 -23352.893,E2 -23352.893} C_VEL
LIN {X 0,Y 187.477,Z 416.877,A -85,B 0,C 180,E1 -23355.419,E2 -23355.419} C_VEL
LIN {X 0,Y 192.058,Z 407.45,A -85,B 0,C 180,E1 -23357.817,E2 -23357.817} C_VEL
LIN {X 0,Y 196.49,Z 396.666,A -85,B 0,C 180,E1 -23359.922,E2 -23359.922} C_VEL
LIN {X 0,Y 200.379,Z 384.993,A -85,B 0,C 180,E1 -23361.698,E2 -23361.698} C_VEL
LIN {X 0,Y 203.494,Z 373.425,A -85,B 0,C 180,E1 -23363.001,E2 -23363.001} C_VEL
LIN {X 0,Y 206.169,Z 360.261,A -85,B 0,C 180,E1 -23364.055,E2 -23364.055} C_VEL
LIN {X 0,Y 207.853,Z 347.827,A -85,B 0,C 180,E1 -23364.725,E2 -23364.725} C_VEL
LIN {X 0,Y 210.301,Z 313.241,A -85,B 0,C 180,E1 -23365.816,E2 -23365.816} C_VEL
LIN {X 0,Y 205.102,Z 303.276,A -85,B 0,C 180,E1 -23368.135,E2 -23368.135} C_VEL
LIN {X 0,Y 199.012,Z 293.191,A -85,B 0,C 180,E1 -23371.094,E2 -23371.094} C_VEL
LIN {X 0,Y 193.055,Z 284.348,A -85,B 0,C 180,E1 -23374.362,E2 -23374.362} C_VEL
LIN {X 0,Y 189.894,Z 279.947,A -85,B 0,C 180,E1 -23376.302,E2 -23376.302} C_VEL
LIN {X 0,Y 186.855,Z 275.851,A -85,B 0,C 180,E1 -23378.342,E2 -23378.342} C_VEL
LIN {X 0,Y 183.667,Z 271.585,A -85,B 0,C 180,E1 -23380.729,E2 -23380.729} C_VEL
LIN {X 0,Y 180.806,Z 268.429,A -85,B 0,C 180,E1 -23383.087,E2 -23383.087} C_VEL
LIN {X 0,Y 179.541,Z 266.327,A -85,B 0,C 180,E1 -23384.315,E2 -23384.315} C_VEL
LIN {X 0,Y 176.888,Z 263.915,A -85,B 0,C 180,E1 -23386.976,E2 -23386.976} C_VEL
LIN {X 0,Y 175.239,Z 260.834,A -85,B 0,C 180,E1 -23389.112,E2 -23389.112} C_VEL
LIN {X 0,Y 172.168,Z 258.479,A -85,B 0,C 180,E1 -23393.554,E2 -23393.554} C_VEL
LIN {X 0,Y 170.94,Z 256.115,A -85,B 0,C 180,E1 -23396.317,E2 -23396.317} C_VEL
LIN {X 0,Y 170.726,Z 255.159,A -85,B 0,C 180,E1 -23397.05,E2 -23397.05} C_VEL
LIN {X 0,Y 169.231,Z 254.553,A -85,B 0,C 180,E1 -23402.38,E2 -23402.38} C_VEL
LIN {X 0,Y 170.386,Z 255.057,A -85,B 0,C 180,E1 -23412.506,E2 -23412.506} C_VEL
LIN {X 0,Y 170.685,Z 256.127,A -85,B 0,C 180,E1 -23413.543,E2 -23413.543} C_VEL
LIN {X 0,Y 172.15,Z 258.871,A -85,B 0,C 180,E1 -23416.91,E2 -23416.91} C_VEL
LIN {X 0,Y 175.32,Z 261.258,A -85,B 0,C 180,E1 -23421.456,E2 -23421.456} C_VEL
LIN {X 0,Y 177.258,Z 264.554,A -85,B 0,C 180,E1 -23423.877,E2 -23423.877} C_VEL
LIN {X 0,Y 180.721,Z 268.84,A -85,B 0,C 180,E1 -23427.308,E2 -23427.308} C_VEL
LIN {X 0,Y 185.476,Z 275.938,A -85,B 0,C 180,E1 -23431.244,E2 -23431.244} C_VEL
LIN {X 0,Y 189.165,Z 281.881,A -85,B 0,C 180,E1 -23433.869,E2 -23433.869} C_VEL
LIN {X 0,Y 192.179,Z 286.975,A -85,B 0,C 180,E1 -23435.811,E2 -23435.811} C_VEL
LIN {X 0,Y 197.196,Z 295.858,A -85,B 0,C 180,E1 -23438.724,E2 -23438.724} C_VEL
LIN {X 0,Y 203.047,Z 307.718,A -85,B 0,C 180,E1 -23441.782,E2 -23441.782} C_VEL
LIN {X 0,Y 207.424,Z 318.108,A -85,B 0,C 180,E1 -23443.91,E2 -23443.91} C_VEL
LIN {X 0,Y 209.46,Z 323.808,A -85,B 0,C 180,E1 -23444.883,E2 -23444.883} C_VEL
LIN {X 0,Y 209.386,Z 328.712,A -85,B 0,C 180,E1 -23445.115,E2 -23445.115} C_VEL
LIN {X 0,Y 207.005,Z 360.877,A -85,B 0,C 180,E1 -23446.11,E2 -23446.11} C_VEL
LIN {X 0,Y 205.072,Z 374.186,A -85,B 0,C 180,E1 -23446.816,E2 -23446.816} C_VEL
LIN {X 0,Y 202.117,Z 387.246,A -85,B 0,C 180,E1 -23447.815,E2 -23447.815} C_VEL
LIN {X 0,Y 198.54,Z 399.065,A -85,B 0,C 180,E1 -23449.09,E2 -23449.09} C_VEL
LIN {X 0,Y 194.846,Z 409.151,A -85,B 0,C 180,E1 -23450.526,E2 -23450.526} C_VEL
LIN {X 0,Y 190.369,Z 419.646,A -85,B 0,C 180,E1 -23452.472,E2 -23452.472} C_VEL
LIN {X 0,Y 185.528,Z 429.469,A -85,B 0,C 180,E1 -23454.848,E2 -23454.848} C_VEL
LIN {X 0,Y 182.752,Z 433.535,A -85,B 0,C 180,E1 -23455.91,E2 -23455.91} C_VEL
LIN {X 0,Y 174.237,Z 441.922,A -85,B 0,C 180,E1 -23458.186,E2 -23458.186} C_VEL
LIN {X 0,Y 169.783,Z 446.192,A -85,B 0,C 180,E1 -23459.814,E2 -23459.814} C_VEL
LIN {X 0,Y 168.167,Z 448.158,A -85,B 0,C 180,E1 -23460.814,E2 -23460.814} C_VEL
LIN {X 0,Y 164.052,Z 454.096,A -85,B 0,C 180,E1 -23464.632,E2 -23464.632} C_VEL
LIN {X 0,Y 160.821,Z 458.213,A -85,B 0,C 180,E1 -23468.192,E2 -23468.192} C_VEL
LIN {X 0,Y 158.261,Z 461.302,A -85,B 0,C 180,E1 -23471.886,E2 -23471.886} C_VEL
LIN {X 0,Y 156.936,Z 462.855,A -85,B 0,C 180,E1 -23474.41,E2 -23474.41} C_VEL
LIN {X 0,Y 155.335,Z 464.703,A -85,B 0,C 180,E1 -23479.569,E2 -23479.569} C_VEL
LIN {X 0,Y 154.844,Z 465.031,A -85,B 0,C 180,E1 -23484.787,E2 -23484.787} C_VEL
LIN {X 0,Y 154.905,Z 464.584,A -85,B 0,C 180,E1 -23487.395,E2 -23487.395} C_VEL
LIN {X 0,Y 155.104,Z 463.726,A -85,B 0,C 180,E1 -23489.995,E2 -23489.995} C_VEL
LIN {X 0,Y 154.875,Z 462.028,A -85,B 0,C 180,E1 -23493.311,E2 -23493.311} C_VEL
LIN {X 0,Y 155.036,Z 458.532,A -85,B 0,C 180,E1 -23497.81,E2 -23497.81} C_VEL
LIN {X 0,Y 155.56,Z 454.338,A -85,B 0,C 180,E1 -23501.724,E2 -23501.724} C_VEL
LIN {X 0,Y 156.955,Z 447.921,A -85,B 0,C 180,E1 -23506.245,E2 -23506.245} C_VEL
LIN {X 0,Y 158.865,Z 440.92,A -85,B 0,C 180,E1 -23510.043,E2 -23510.043} C_VEL
LIN {X 0,Y 160.456,Z 435.261,A -85,B 0,C 180,E1 -23512.528,E2 -23512.528} C_VEL
LIN {X 0,Y 162.97,Z 426.94,A -85,B 0,C 180,E1 -23515.539,E2 -23515.539} C_VEL
LIN {X 0,Y 165.797,Z 416.735,A -85,B 0,C 180,E1 -23518.474,E2 -23518.474} C_VEL
LIN {X 0,Y 168.081,Z 408.017,A -85,B 0,C 180,E1 -23520.455,E2 -23520.455} C_VEL
LIN {X 0,Y 170.642,Z 397.369,A -85,B 0,C 180,E1 -23522.363,E2 -23522.363} C_VEL
LIN {X 0,Y 173.179,Z 384.524,A -85,B 0,C 180,E1 -23524.084,E2 -23524.084} C_VEL
LIN {X 0,Y 175.08,Z 371.587,A -85,B 0,C 180,E1 -23525.321,E2 -23525.321} C_VEL
LIN {X 0,Y 176.331,Z 358.885,A -85,B 0,C 180,E1 -23526.086,E2 -23526.086} C_VEL
LIN {X 0,Y 178.386,Z 316.242,A -85,B 0,C 180,E1 -23527.713,E2 -23527.713} C_VEL
LIN {X 0,Y 176.422,Z 292.721,A -85,B 0,C 180,E1 -23529.257,E2 -23529.257} C_VEL
LIN {X 0,Y 171.025,Z 278.407,A -85,B 0,C 180,E1 -23531.218,E2 -23531.218} C_VEL
LIN {X 0,Y 165.713,Z 266.573,A -85,B 0,C 180,E1 -23533.203,E2 -23533.203} C_VEL
LIN {X 0,Y 159.881,Z 255.547,A -85,B 0,C 180,E1 -23535.487,E2 -23535.487} C_VEL
LIN {X 0,Y 157.496,Z 251.059,A -85,B 0,C 180,E1 -23536.571,E2 -23536.571} C_VEL
LIN {X 0,Y 157.223,Z 249.9,A -85,B 0,C 180,E1 -23537.382,E2 -23537.382} C_VEL
LIN {X 0,Y 157.262,Z 249.895,A -85,B 0,C 180,E1 -23543.538,E2 -23543.538} C_VEL
LIN {X 0,Y 157.27,Z 249.896,A -85,B 0,C 180,E1 -23548.092,E2 -23548.092} C_VEL
LIN {X 0,Y 157.297,Z 249.888,A -85,B 0,C 180,E1 -23553.462,E2 -23553.462} C_VEL
LIN {X 0,Y 157.421,Z 249.876,A -85,B 0,C 180,E1 -23559.613,E2 -23559.613} C_VEL
LIN {X 0,Y 157.418,Z 249.876,A -85,B 0,C 180,E1 -23564.462,E2 -23564.462} C_VEL
LIN {X 0,Y 157.659,Z 249.846,A -85,B 0,C 180,E1 -23569.729,E2 -23569.729} C_VEL
LIN {X 0,Y 157.735,Z 249.827,A -85,B 0,C 180,E1 -23572.319,E2 -23572.319} C_VEL
LIN {X 0,Y 158.216,Z 249.745,A -85,B 0,C 180,E1 -23580,E2 -23580} C_VEL
LIN {X 0,Y 157.73,Z 249.835,A -85,B 0,C 180,E1 -23587.682,E2 -23587.682} C_VEL
LIN {X 0,Y 157.601,Z 249.838,A -85,B 0,C 180,E1 -23591.223,E2 -23591.223} C_VEL
LIN {X 0,Y 157.378,Z 249.844,A -85,B 0,C 180,E1 -23595.542,E2 -23595.542} C_VEL
LIN {X 0,Y 157.284,Z 249.892,A -85,B 0,C 180,E1 -23600.945,E2 -23600.945} C_VEL
LIN {X 0,Y 157.286,Z 249.893,A -85,B 0,C 180,E1 -23606.685,E2 -23606.685} C_VEL
LIN {X 0,Y 157.254,Z 249.896,A -85,B 0,C 180,E1 -23612.433,E2 -23612.433} C_VEL
LIN {X 0,Y 157.263,Z 249.895,A -85,B 0,C 180,E1 -23616.462,E2 -23616.462} C_VEL
LIN {X 0,Y 157.217,Z 249.898,A -85,B 0,C 180,E1 -23622.109,E2 -23622.109} C_VEL
LIN {X 0,Y 157.195,Z 249.889,A -85,B 0,C 180,E1 -23627.896,E2 -23627.896} C_VEL
LIN {X 0,Y 157.246,Z 249.879,A -85,B 0,C 180,E1 -23633.563,E2 -23633.563} C_VEL
LIN {X 0,Y 157.256,Z 249.948,A -85,B 0,C 180,E1 -23635.087,E2 -23635.087} C_VEL
LIN {X 0,Y 158.388,Z 252.95,A -85,B 0,C 180,E1 -23635.623,E2 -23635.623} C_VEL
LIN {X 0,Y 160.112,Z 255.089,A -85,B 0,C 180,E1 -23636.278,E2 -23636.278} C_VEL
LIN {X 0,Y 167.096,Z 266.393,A -85,B 0,C 180,E1 -23638.881,E2 -23638.881} C_VEL
LIN {X 0,Y 174.5,Z 280.271,A -85,B 0,C 180,E1 -23641.426,E2 -23641.426} C_VEL
LIN {X 0,Y 179.561,Z 291.844,A -85,B 0,C 180,E1 -23643.103,E2 -23643.103} C_VEL
LIN {X 0,Y 176.564,Z 347.331,A -85,B 0,C 180,E1 -23645.174,E2 -23645.174} C_VEL
LIN {X 0,Y 175.186,Z 360.546,A -85,B 0,C 180,E1 -23646.079,E2 -23646.079} C_VEL
LIN {X 0,Y 173.684,Z 371.729,A -85,B 0,C 180,E1 -23647.243,E2 -23647.243} C_VEL
LIN {X 0,Y 171.615,Z 384.111,A -85,B 0,C 180,E1 -23649.009,E2 -23649.009} C_VEL
LIN {X 0,Y 168.86,Z 395.795,A -85,B 0,C 180,E1 -23651.189,E2 -23651.189} C_VEL
LIN {X 0,Y 166.17,Z 406.26,A -85,B 0,C 180,E1 -23653.734,E2 -23653.734} C_VEL
LIN {X 0,Y 163.633,Z 414.841,A -85,B 0,C 180,E1 -23656.342,E2 -23656.342} C_VEL
LIN {X 0,Y 161.372,Z 422.722,A -85,B 0,C 180,E1 -23659.339,E2 -23659.339} C_VEL
LIN {X 0,Y 159,Z 430.449,A -85,B 0,C 180,E1 -23663.024,E2 -23663.024} C_VEL
LIN {X 0,Y 157.511,Z 435.723,A -85,B 0,C 180,E1 -23666.168,E2 -23666.168} C_VEL
LIN {X 0,Y 156.212,Z 440.845,A -85,B 0,C 180,E1 -23670.005,E2 -23670.005} C_VEL
LIN {X 0,Y 155.472,Z 444.826,A -85,B 0,C 180,E1 -23673.893,E2 -23673.893} C_VEL
LIN {X 0,Y 154.845,Z 447.802,A -85,B 0,C 180,E1 -23677.83,E2 -23677.83} C_VEL
LIN {X 0,Y 154.733,Z 449.219,A -85,B 0,C 180,E1 -23680.472,E2 -23680.472} C_VEL
LIN {X 0,Y 155.161,Z 450.865,A -85,B 0,C 180,E1 -23685.773,E2 -23685.773} C_VEL
LIN {X 0,Y 155.77,Z 451.066,A -85,B 0,C 180,E1 -23688.651,E2 -23688.651} C_VEL
LIN {X 0,Y 157.497,Z 450.243,A -85,B 0,C 180,E1 -23693.681,E2 -23693.681} C_VEL
LIN {X 0,Y 158.8,Z 449.229,A -85,B 0,C 180,E1 -23696.27,E2 -23696.27} C_VEL
LIN {X 0,Y 160.384,Z 447.75,A -85,B 0,C 180,E1 -23698.82,E2 -23698.82} C_VEL
LIN {X 0,Y 163.261,Z 444.703,A -85,B 0,C 180,E1 -23702.556,E2 -23702.556} C_VEL
LIN {X 0,Y 166.76,Z 440.547,A -85,B 0,C 180,E1 -23706.16,E2 -23706.16} C_VEL
LIN {X 0,Y 171.559,Z 434.132,A -85,B 0,C 180,E1 -23710.182,E2 -23710.182} C_VEL
LIN {X 0,Y 176.249,Z 427.168,A -85,B 0,C 180,E1 -23713.406,E2 -23713.406} C_VEL
LIN {X 0,Y 180.582,Z 419.801,A -85,B 0,C 180,E1 -23716.054,E2 -23716.054} C_VEL
LIN {X 0,Y 185.275,Z 410.925,A -85,B 0,C 180,E1 -23718.519,E2 -23718.519} C_VEL
LIN {X 0,Y 189.749,Z 401.13,A -85,B 0,C 180,E1 -23720.639,E2 -23720.639} C_VEL
LIN {X 0,Y 193.924,Z 390.202,A -85,B 0,C 180,E1 -23722.486,E2 -23722.486} C_VEL
LIN {X 0,Y 197.501,Z 378.18,A -85,B 0,C 180,E1 -23724.051,E2 -23724.051} C_VEL
LIN {X 0,Y 200.617,Z 365.311,A -85,B 0,C 180,E1 -23725.211,E2 -23725.211} C_VEL
LIN {X 0,Y 202.729,Z 352.345,A -85,B 0,C 180,E1 -23726.034,E2 -23726.034} C_VEL
LIN {X 0,Y 204.154,Z 336.959,A -85,B 0,C 180,E1 -23726.595,E2 -23726.595} C_VEL
LIN {X 0,Y 205.575,Z 315.889,A -85,B 0,C 180,E1 -23727.262,E2 -23727.262} C_VEL
LIN {X 0,Y 200.714,Z 306.758,A -85,B 0,C 180,E1 -23729.579,E2 -23729.579} C_VEL
LIN {X 0,Y 195.299,Z 297.654,A -85,B 0,C 180,E1 -23732.407,E2 -23732.407} C_VEL
LIN {X 0,Y 189.986,Z 289.643,A -85,B 0,C 180,E1 -23735.524,E2 -23735.524} C_VEL
LIN {X 0,Y 187.31,Z 285.773,A -85,B 0,C 180,E1 -23737.272,E2 -23737.272} C_VEL
LIN {X 0,Y 184.509,Z 281.932,A -85,B 0,C 180,E1 -23739.26,E2 -23739.26} C_VEL
LIN {X 0,Y 181.637,Z 277.991,A -85,B 0,C 180,E1 -23741.53,E2 -23741.53} C_VEL
LIN {X 0,Y 178.795,Z 274.563,A -85,B 0,C 180,E1 -23744.029,E2 -23744.029} C_VEL
LIN {X 0,Y 177.808,Z 272.952,A -85,B 0,C 180,E1 -23745.039,E2 -23745.039} C_VEL
LIN {X 0,Y 175.191,Z 270.307,A -85,B 0,C 180,E1 -23747.842,E2 -23747.842} C_VEL
LIN {X 0,Y 173.85,Z 267.692,A -85,B 0,C 180,E1 -23749.689,E2 -23749.689} C_VEL
LIN {X 0,Y 171.011,Z 265.311,A -85,B 0,C 180,E1 -23754.029,E2 -23754.029} C_VEL
LIN {X 0,Y 169.807,Z 262.926,A -85,B 0,C 180,E1 -23756.923,E2 -23756.923} C_VEL
LIN {X 0,Y 169.617,Z 262.075,A -85,B 0,C 180,E1 -23757.625,E2 -23757.625} C_VEL
LIN {X 0,Y 168.359,Z 261.575,A -85,B 0,C 180,E1 -23762.392,E2 -23762.392} C_VEL
LIN {X 0,Y 169.312,Z 262.056,A -85,B 0,C 180,E1 -23771.978,E2 -23771.978} C_VEL
LIN {X 0,Y 170.826,Z 265.547,A -85,B 0,C 180,E1 -23776.123,E2 -23776.123} C_VEL
LIN {X 0,Y 173.973,Z 268.179,A -85,B 0,C 180,E1 -23780.944,E2 -23780.944} C_VEL
LIN {X 0,Y 175.991,Z 271.512,A -85,B 0,C 180,E1 -23783.537,E2 -23783.537} C_VEL
LIN {X 0,Y 178.887,Z 275.317,A -85,B 0,C 180,E1 -23786.544,E2 -23786.544} C_VEL
LIN {X 0,Y 183.189,Z 281.962,A -85,B 0,C 180,E1 -23790.314,E2 -23790.314} C_VEL
LIN {X 0,Y 186.828,Z 288.095,A -85,B 0,C 180,E1 -23793.056,E2 -23793.056} C_VEL
LIN {X 0,Y 189.654,Z 293.071,A -85,B 0,C 180,E1 -23794.975,E2 -23794.975} C_VEL
LIN {X 0,Y 193.94,Z 300.91,A -85,B 0,C 180,E1 -23797.614,E2 -23797.614} C_VEL
LIN {X 0,Y 199.471,Z 312.529,A -85,B 0,C 180,E1 -23800.697,E2 -23800.697} C_VEL
LIN {X 0,Y 204.075,Z 323.884,A -85,B 0,C 180,E1 -23803.072,E2 -23803.072} C_VEL
LIN {X 0,Y 204.953,Z 326.359,A -85,B 0,C 180,E1 -23803.516,E2 -23803.516} C_VEL
LIN {X 0,Y 202.364,Z 360.756,A -85,B 0,C 180,E1 -23804.605,E2 -23804.605} C_VEL
LIN {X 0,Y 200.285,Z 374.371,A -85,B 0,C 180,E1 -23805.334,E2 -23805.334} C_VEL
LIN {X 0,Y 197.241,Z 387.297,A -85,B 0,C 180,E1 -23806.341,E2 -23806.341} C_VEL
LIN {X 0,Y 193.251,Z 399.82,A -85,B 0,C 180,E1 -23807.717,E2 -23807.717} C_VEL
LIN {X 0,Y 189.451,Z 409.706,A -85,B 0,C 180,E1 -23809.169,E2 -23809.169} C_VEL
LIN {X 0,Y 184.804,Z 420.051,A -85,B 0,C 180,E1 -23811.134,E2 -23811.134} C_VEL
LIN {X 0,Y 179.711,Z 429.837,A -85,B 0,C 180,E1 -23813.584,E2 -23813.584} C_VEL
LIN {X 0,Y 174.684,Z 438.417,A -85,B 0,C 180,E1 -23816.412,E2 -23816.412} C_VEL
LIN {X 0,Y 169.872,Z 445.729,A -85,B 0,C 180,E1 -23819.547,E2 -23819.547} C_VEL
LIN {X 0,Y 168.167,Z 448.158,A -85,B 0,C 180,E1 -23820.814,E2 -23820.814} C_VEL
LIN {X 0,Y 165.628,Z 450.992,A -85,B 0,C 180,E1 -23822.373,E2 -23822.373} C_VEL
LIN {X 0,Y 159.996,Z 455.048,A -85,B 0,C 180,E1 -23824.871,E2 -23824.871} C_VEL
LIN {X 0,Y 155.535,Z 457.792,A -85,B 0,C 180,E1 -23827.051,E2 -23827.051} C_VEL
LIN {X 0,Y 153.016,Z 459.569,A -85,B 0,C 180,E1 -23828.93,E2 -23828.93} C_VEL
LIN {X 0,Y 152.455,Z 460.049,A -85,B 0,C 180,E1 -23829.61,E2 -23829.61} C_VEL
LIN {X 0,Y 150.072,Z 462.627,A -85,B 0,C 180,E1 -23833.677,E2 -23833.677} C_VEL
LIN {X 0,Y 148.329,Z 464.414,A -85,B 0,C 180,E1 -23839.071,E2 -23839.071} C_VEL
LIN {X 0,Y 147.75,Z 464.679,A -85,B 0,C 180,E1 -23844.536,E2 -23844.536} C_VEL
LIN {X 0,Y 147.824,Z 464.19,A -85,B 0,C 180,E1 -23847.27,E2 -23847.27} C_VEL
LIN {X 0,Y 148.005,Z 463.305,A -85,B 0,C 180,E1 -23849.995,E2 -23849.995} C_VEL
LIN {X 0,Y 147.794,Z 461.823,A -85,B 0,C 180,E1 -23853.026,E2 -23853.026} C_VEL
LIN {X 0,Y 147.896,Z 459.169,A -85,B 0,C 180,E1 -23856.817,E2 -23856.817} C_VEL
LIN {X 0,Y 148.331,Z 455.287,A -85,B 0,C 180,E1 -23860.919,E2 -23860.919} C_VEL
LIN {X 0,Y 149.317,Z 450.246,A -85,B 0,C 180,E1 -23864.996,E2 -23864.996} C_VEL
LIN {X 0,Y 151.127,Z 443.913,A -85,B 0,C 180,E1 -23868.99,E2 -23868.99} C_VEL
LIN {X 0,Y 153.456,Z 435.943,A -85,B 0,C 180,E1 -23872.902,E2 -23872.902} C_VEL
LIN {X 0,Y 155.385,Z 429.594,A -85,B 0,C 180,E1 -23875.438,E2 -23875.438} C_VEL
LIN {X 0,Y 158.324,Z 420.051,A -85,B 0,C 180,E1 -23878.494,E2 -23878.494} C_VEL
LIN {X 0,Y 160.852,Z 410.727,A -85,B 0,C 180,E1 -23880.881,E2 -23880.881} C_VEL
LIN {X 0,Y 163.886,Z 399.23,A -85,B 0,C 180,E1 -23883.136,E2 -23883.136} C_VEL
LIN {X 0,Y 166.504,Z 387.219,A -85,B 0,C 180,E1 -23884.913,E2 -23884.913} C_VEL
LIN {X 0,Y 168.533,Z 374.576,A -85,B 0,C 180,E1 -23886.263,E2 -23886.263} C_VEL
LIN {X 0,Y 170.084,Z 361.581,A -85,B 0,C 180,E1 -23887.17,E2 -23887.17} C_VEL
LIN {X 0,Y 172.427,Z 316.858,A -85,B 0,C 180,E1 -23888.957,E2 -23888.957} C_VEL
LIN {X 0,Y 170.656,Z 295.002,A -85,B 0,C 180,E1 -23890.459,E2 -23890.459} C_VEL
LIN {X 0,Y 165.815,Z 281.945,A -85,B 0,C 180,E1 -23892.347,E2 -23892.347} C_VEL
LIN {X 0,Y 160.388,Z 269.603,A -85,B 0,C 180,E1 -23894.53,E2 -23894.53} C_VEL
LIN {X 0,Y 155.112,Z 259.684,A -85,B 0,C 180,E1 -23896.741,E2 -23896.741} C_VEL
LIN {X 0,Y 152.611,Z 255.268,A -85,B 0,C 180,E1 -23897.852,E2 -23897.852} C_VEL
LIN {X 0,Y 150.83,Z 253.037,A -85,B 0,C 180,E1 -23898.62,E2 -23898.62} C_VEL
LIN {X 0,Y 150.168,Z 250.782,A -85,B 0,C 180,E1 -23899.064,E2 -23899.064} C_VEL
LIN {X 0,Y 150.197,Z 250.775,A -85,B 0,C 180,E1 -23902.683,E2 -23902.683} C_VEL
LIN {X 0,Y 150.194,Z 250.777,A -85,B 0,C 180,E1 -23907.363,E2 -23907.363} C_VEL
LIN {X 0,Y 150.22,Z 250.771,A -85,B 0,C 180,E1 -23912.715,E2 -23912.715} C_VEL
LIN {X 0,Y 150.364,Z 250.755,A -85,B 0,C 180,E1 -23919.166,E2 -23919.166} C_VEL
LIN {X 0,Y 150.335,Z 250.759,A -85,B 0,C 180,E1 -23923.711,E2 -23923.711} C_VEL
LIN {X 0,Y 150.58,Z 250.728,A -85,B 0,C 180,E1 -23929.24,E2 -23929.24} C_VEL
LIN {X 0,Y 150.673,Z 250.708,A -85,B 0,C 180,E1 -23931.956,E2 -23931.956} C_VEL
LIN {X 0,Y 151.176,Z 250.62,A -85,B 0,C 180,E1 -23940,E2 -23940} C_VEL
LIN {X 0,Y 150.668,Z 250.715,A -85,B 0,C 180,E1 -23948.044,E2 -23948.044} C_VEL
LIN {X 0,Y 150.544,Z 250.712,A -85,B 0,C 180,E1 -23951.427,E2 -23951.427} C_VEL
LIN {X 0,Y 150.283,Z 250.732,A -85,B 0,C 180,E1 -23956.296,E2 -23956.296} C_VEL
LIN {X 0,Y 150.258,Z 250.768,A -85,B 0,C 180,E1 -23960.727,E2 -23960.727} C_VEL
LIN {X 0,Y 150.218,Z 250.771,A -85,B 0,C 180,E1 -23967.284,E2 -23967.284} C_VEL
LIN {X 0,Y 150.194,Z 250.774,A -85,B 0,C 180,E1 -23972.638,E2 -23972.638} C_VEL
LIN {X 0,Y 150.194,Z 250.775,A -85,B 0,C 180,E1 -23977.468,E2 -23977.468} C_VEL
LIN {X 0,Y 150.157,Z 250.778,A -85,B 0,C 180,E1 -23981.522,E2 -23981.522} C_VEL
LIN {X 0,Y 150.12,Z 250.757,A -85,B 0,C 180,E1 -23985.406,E2 -23985.406} C_VEL
LIN {X 0,Y 150.134,Z 250.779,A -85,B 0,C 180,E1 -23989.065,E2 -23989.065} C_VEL
LIN {X 0,Y 150.163,Z 250.775,A -85,B 0,C 180,E1 -23992.717,E2 -23992.717} C_VEL
LIN {X 0,Y 151.173,Z 253.597,A -85,B 0,C 180,E1 -23993.263,E2 -23993.263} C_VEL
LIN {X 0,Y 153.235,Z 256.111,A -85,B 0,C 180,E1 -23994.138,E2 -23994.138} C_VEL
LIN {X 0,Y 155.308,Z 259.326,A -85,B 0,C 180,E1 -23995.025,E2 -23995.025} C_VEL
LIN {X 0,Y 162.232,Z 270.461,A -85,B 0,C 180,E1 -23997.773,E2 -23997.773} C_VEL
LIN {X 0,Y 169.497,Z 284.353,A -85,B 0,C 180,E1 -24000.44,E2 -24000.44} C_VEL
LIN {X 0,Y 173.506,Z 293.453,A -85,B 0,C 180,E1 -24001.852,E2 -24001.852} C_VEL
LIN {X 0,Y 170.533,Z 347.733,A -85,B 0,C 180,E1 -24003.952,E2 -24003.952} C_VEL
LIN {X 0,Y 169.068,Z 361.117,A -85,B 0,C 180,E1 -24004.895,E2 -24004.895} C_VEL
LIN {X 0,Y 167.233,Z 374,A -85,B 0,C 180,E1 -24006.313,E2 -24006.313} C_VEL
LIN {X 0,Y 165.034,Z 385.83,A -85,B 0,C 180,E1 -24008.13,E2 -24008.13} C_VEL
LIN {X 0,Y 162.183,Z 397.25,A -85,B 0,C 180,E1 -24010.384,E2 -24010.384} C_VEL
LIN {X 0,Y 159.403,Z 407.519,A -85,B 0,C 180,E1 -24013.023,E2 -24013.023} C_VEL
LIN {X 0,Y 156.778,Z 415.94,A -85,B 0,C 180,E1 -24015.733,E2 -24015.733} C_VEL
LIN {X 0,Y 154.023,Z 425.03,A -85,B 0,C 180,E1 -24019.49,E2 -24019.49} C_VEL
LIN {X 0,Y 151.584,Z 432.388,A -85,B 0,C 180,E1 -24023.35,E2 -24023.35} C_VEL
LIN {X 0,Y 149.957,Z 438.267,A -85,B 0,C 180,E1 -24027.319,E2 -24027.319} C_VEL
LIN {X 0,Y 148.795,Z 442.918,A -85,B 0,C 180,E1 -24031.358,E2 -24031.358} C_VEL
LIN {X 0,Y 148.107,Z 446.476,A -85,B 0,C 180,E1 -24035.45,E2 -24035.45} C_VEL
LIN {X 0,Y 147.725,Z 448.299,A -85,B 0,C 180,E1 -24038.21,E2 -24038.21} C_VEL
LIN {X 0,Y 147.625,Z 449.678,A -85,B 0,C 180,E1 -24040.982,E2 -24040.982} C_VEL
LIN {X 0,Y 147.758,Z 450.662,A -85,B 0,C 180,E1 -24043.762,E2 -24043.762} C_VEL
LIN {X 0,Y 148.181,Z 451.248,A -85,B 0,C 180,E1 -24046.537,E2 -24046.537} C_VEL
LIN {X 0,Y 148.818,Z 451.393,A -85,B 0,C 180,E1 -24049.307,E2 -24049.307} C_VEL
LIN {X 0,Y 150.823,Z 450.489,A -85,B 0,C 180,E1 -24054.798,E2 -24054.798} C_VEL
LIN {X 0,Y 153.694,Z 448.195,A -85,B 0,C 180,E1 -24059.678,E2 -24059.678} C_VEL
LIN {X 0,Y 157.13,Z 444.761,A -85,B 0,C 180,E1 -24063.995,E2 -24063.995} C_VEL
LIN {X 0,Y 160.893,Z 440.522,A -85,B 0,C 180,E1 -24067.702,E2 -24067.702} C_VEL
LIN {X 0,Y 165.258,Z 435.038,A -85,B 0,C 180,E1 -24071.238,E2 -24071.238} C_VEL
LIN {X 0,Y 170.194,Z 428.126,A -85,B 0,C 180,E1 -24074.588,E2 -24074.588} C_VEL
LIN {X 0,Y 174.651,Z 421.015,A -85,B 0,C 180,E1 -24077.256,E2 -24077.256} C_VEL
LIN {X 0,Y 179.519,Z 412.378,A -85,B 0,C 180,E1 -24079.765,E2 -24079.765} C_VEL
LIN {X 0,Y 184.14,Z 402.813,A -85,B 0,C 180,E1 -24081.923,E2 -24081.923} C_VEL
LIN {X 0,Y 188.416,Z 392.327,A -85,B 0,C 180,E1 -24083.765,E2 -24083.765} C_VEL
LIN {X 0,Y 192.189,Z 380.734,A -85,B 0,C 180,E1 -24085.363,E2 -24085.363} C_VEL
LIN {X 0,Y 195.35,Z 368.873,A -85,B 0,C 180,E1 -24086.516,E2 -24086.516} C_VEL
LIN {X 0,Y 197.868,Z 355.33,A -85,B 0,C 180,E1 -24087.449,E2 -24087.449} C_VEL
LIN {X 0,Y 199.323,Z 342.61,A -85,B 0,C 180,E1 -24087.995,E2 -24087.995} C_VEL
LIN {X 0,Y 201.028,Z 318.949,A -85,B 0,C 180,E1 -24088.738,E2 -24088.738} C_VEL
LIN {X 0,Y 195.859,Z 309.159,A -85,B 0,C 180,E1 -24091.415,E2 -24091.415} C_VEL
LIN {X 0,Y 190.519,Z 300.216,A -85,B 0,C 180,E1 -24094.48,E2 -24094.48} C_VEL
LIN {X 0,Y 185.134,Z 292.095,A -85,B 0,C 180,E1 -24098.02,E2 -24098.02} C_VEL
LIN {X 0,Y 182.299,Z 288.098,A -85,B 0,C 180,E1 -24100.139,E2 -24100.139} C_VEL
LIN {X 0,Y 179.567,Z 284.309,A -85,B 0,C 180,E1 -24102.416,E2 -24102.416} C_VEL
LIN {X 0,Y 176.775,Z 280.577,A -85,B 0,C 180,E1 -24105.06,E2 -24105.06} C_VEL
LIN {X 0,Y 176.04,Z 279.498,A -85,B 0,C 180,E1 -24105.846,E2 -24105.846} C_VEL
LIN {X 0,Y 173.511,Z 276.64,A -85,B 0,C 180,E1 -24108.759,E2 -24108.759} C_VEL
LIN {X 0,Y 172.415,Z 274.47,A -85,B 0,C 180,E1 -24110.367,E2 -24110.367} C_VEL
LIN {X 0,Y 169.721,Z 271.981,A -85,B 0,C 180,E1 -24114.803,E2 -24114.803} C_VEL
LIN {X 0,Y 168.637,Z 269.467,A -85,B 0,C 180,E1 -24117.761,E2 -24117.761} C_VEL
LIN {X 0,Y 168.526,Z 268.996,A -85,B 0,C 180,E1 -24118.207,E2 -24118.207} C_VEL
LIN {X 0,Y 167.264,Z 268.693,A -85,B 0,C 180,E1 -24124.82,E2 -24124.82} C_VEL
LIN {X 0,Y 168.366,Z 269.157,A -85,B 0,C 180,E1 -24131.813,E2 -24131.813} C_VEL
LIN {X 0,Y 169.441,Z 272.027,A -85,B 0,C 180,E1 -24135.101,E2 -24135.101} C_VEL
LIN {X 0,Y 172.576,Z 274.991,A -85,B 0,C 180,E1 -24140.33,E2 -24140.33} C_VEL
LIN {X 0,Y 177.104,Z 281.808,A -85,B 0,C 180,E1 -24145.782,E2 -24145.782} C_VEL
LIN {X 0,Y 181.025,Z 288.15,A -85,B 0,C 180,E1 -24149.423,E2 -24149.423} C_VEL
LIN {X 0,Y 184.428,Z 294.129,A -85,B 0,C 180,E1 -24152.146,E2 -24152.146} C_VEL
LIN {X 0,Y 187.263,Z 299.364,A -85,B 0,C 180,E1 -24154.183,E2 -24154.183} C_VEL
LIN {X 0,Y 191.212,Z 306.998,A -85,B 0,C 180,E1 -24156.757,E2 -24156.757} C_VEL
LIN {X 0,Y 196.156,Z 317.785,A -85,B 0,C 180,E1 -24159.677,E2 -24159.677} C_VEL
LIN {X 0,Y 200.32,Z 328.543,A -85,B 0,C 180,E1 -24161.973,E2 -24161.973} C_VEL
LIN {X 0,Y 199.632,Z 339.062,A -85,B 0,C 180,E1 -24162.329,E2 -24162.329} C_VEL
LIN {X 0,Y 197.744,Z 361.574,A -85,B 0,C 180,E1 -24163.07,E2 -24163.07} C_VEL
LIN {X 0,Y 195.54,Z 375.092,A -85,B 0,C 180,E1 -24163.816,E2 -24163.816} C_VEL
LIN {X 0,Y 192.496,Z 387.337,A -85,B 0,C 180,E1 -24164.793,E2 -24164.793} C_VEL
LIN {X 0,Y 188.675,Z 398.996,A -85,B 0,C 180,E1 -24166.071,E2 -24166.071} C_VEL
LIN {X 0,Y 184.712,Z 408.975,A -85,B 0,C 180,E1 -24167.518,E2 -24167.518} C_VEL
LIN {X 0,Y 179.92,Z 419.385,A -85,B 0,C 180,E1 -24169.503,E2 -24169.503} C_VEL
LIN {X 0,Y 175.297,Z 427.919,A -85,B 0,C 180,E1 -24171.579,E2 -24171.579} C_VEL
LIN {X 0,Y 170.577,Z 435.805,A -85,B 0,C 180,E1 -24174.046,E2 -24174.046} C_VEL
LIN {X 0,Y 165.364,Z 443.546,A -85,B 0,C 180,E1 -24177.187,E2 -24177.187} C_VEL
LIN {X 0,Y 161.504,Z 448.852,A -85,B 0,C 180,E1 -24179.969,E2 -24179.969} C_VEL
LIN {X 0,Y 157.633,Z 454.039,A -85,B 0,C 180,E1 -24183.52,E2 -24183.52} C_VEL
LIN {X 0,Y 154.216,Z 458.094,A -85,B 0,C 180,E1 -24187.206,E2 -24187.206} C_VEL
LIN {X 0,Y 152.455,Z 460.049,A -85,B 0,C 180,E1 -24189.61,E2 -24189.61} C_VEL
LIN {X 0,Y 150.499,Z 461.531,A -85,B 0,C 180,E1 -24191.65,E2 -24191.65} C_VEL
LIN {X 0,Y 145.982,Z 463.245,A -85,B 0,C 180,E1 -24195,E2 -24195} C_VEL
LIN {X 0,Y 142.624,Z 464.026,A -85,B 0,C 180,E1 -24197.843,E2 -24197.843} C_VEL
LIN {X 0,Y 141.096,Z 464.335,A -85,B 0,C 180,E1 -24200.148,E2 -24200.148} C_VEL
LIN {X 0,Y 140.895,Z 464.379,A -85,B 0,C 180,E1 -24200.944,E2 -24200.944} C_VEL
LIN {X 0,Y 140.681,Z 464.313,A -85,B 0,C 180,E1 -24204.261,E2 -24204.261} C_VEL
LIN {X 0,Y 140.736,Z 463.795,A -85,B 0,C 180,E1 -24207.132,E2 -24207.132} C_VEL
LIN {X 0,Y 140.908,Z 462.883,A -85,B 0,C 180,E1 -24209.995,E2 -24209.995} C_VEL
LIN {X 0,Y 140.735,Z 461.537,A -85,B 0,C 180,E1 -24212.857,E2 -24212.857} C_VEL
LIN {X 0,Y 140.814,Z 458.659,A -85,B 0,C 180,E1 -24217.162,E2 -24217.162} C_VEL
LIN {X 0,Y 141.326,Z 454.716,A -85,B 0,C 180,E1 -24221.467,E2 -24221.467} C_VEL
LIN {X 0,Y 142.682,Z 448.622,A -85,B 0,C 180,E1 -24226.445,E2 -24226.445} C_VEL
LIN {X 0,Y 144.729,Z 441.929,A -85,B 0,C 180,E1 -24230.606,E2 -24230.606} C_VEL
LIN {X 0,Y 146.745,Z 435.44,A -85,B 0,C 180,E1 -24233.844,E2 -24233.844} C_VEL
LIN {X 0,Y 149.599,Z 426.874,A -85,B 0,C 180,E1 -24237.252,E2 -24237.252} C_VEL
LIN {X 0,Y 152.685,Z 416.806,A -85,B 0,C 180,E1 -24240.41,E2 -24240.41} C_VEL
LIN {X 0,Y 155.163,Z 408.204,A -85,B 0,C 180,E1 -24242.529,E2 -24242.529} C_VEL
LIN {X 0,Y 157.941,Z 397.803,A -85,B 0,C 180,E1 -24244.556,E2 -24244.556} C_VEL
LIN {X 0,Y 160.683,Z 385.332,A -85,B 0,C 180,E1 -24246.374,E2 -24246.374} C_VEL
LIN {X 0,Y 162.775,Z 372.617,A -85,B 0,C 180,E1 -24247.705,E2 -24247.705} C_VEL
LIN {X 0,Y 164.306,Z 359.295,A -85,B 0,C 180,E1 -24248.601,E2 -24248.601} C_VEL
LIN {X 0,Y 166.534,Z 317.749,A -85,B 0,C 180,E1 -24250.276,E2 -24250.276} C_VEL
LIN {X 0,Y 165.051,Z 297.502,A -85,B 0,C 180,E1 -24251.712,E2 -24251.712} C_VEL
LIN {X 0,Y 160.785,Z 285.715,A -85,B 0,C 180,E1 -24253.504,E2 -24253.504} C_VEL
LIN {X 0,Y 155.617,Z 273.706,A -85,B 0,C 180,E1 -24255.735,E2 -24255.735} C_VEL
LIN {X 0,Y 150.757,Z 264.314,A -85,B 0,C 180,E1 -24257.922,E2 -24257.922} C_VEL
LIN {X 0,Y 148.536,Z 260.481,A -85,B 0,C 180,E1 -24258.967,E2 -24258.967} C_VEL
LIN {X 0,Y 146.322,Z 257.112,A -85,B 0,C 180,E1 -24260.028,E2 -24260.028} C_VEL
LIN {X 0,Y 143.803,Z 254.008,A -85,B 0,C 180,E1 -24261.249,E2 -24261.249} C_VEL
LIN {X 0,Y 143.118,Z 251.661,A -85,B 0,C 180,E1 -24261.77,E2 -24261.77} C_VEL
LIN {X 0,Y 143.161,Z 251.652,A -85,B 0,C 180,E1 -24267.316,E2 -24267.316} C_VEL
LIN {X 0,Y 143.166,Z 251.652,A -85,B 0,C 180,E1 -24272.06,E2 -24272.06} C_VEL
LIN {X 0,Y 143.286,Z 251.635,A -85,B 0,C 180,E1 -24278.708,E2 -24278.708} C_VEL
LIN {X 0,Y 143.284,Z 251.635,A -85,B 0,C 180,E1 -24282.885,E2 -24282.885} C_VEL
LIN {X 0,Y 143.506,Z 251.607,A -85,B 0,C 180,E1 -24288.703,E2 -24288.703} C_VEL
LIN {X 0,Y 143.595,Z 251.591,A -85,B 0,C 180,E1 -24291.557,E2 -24291.557} C_VEL
LIN {X 0,Y 144.134,Z 251.495,A -85,B 0,C 180,E1 -24300,E2 -24300} C_VEL
LIN {X 0,Y 143.59,Z 251.597,A -85,B 0,C 180,E1 -24308.444,E2 -24308.444} C_VEL
LIN {X 0,Y 143.469,Z 251.589,A -85,B 0,C 180,E1 -24311.611,E2 -24311.611} C_VEL
LIN {X 0,Y 143.224,Z 251.62,A -85,B 0,C 180,E1 -24317.123,E2 -24317.123} C_VEL
LIN {X 0,Y 143.197,Z 251.646,A -85,B 0,C 180,E1 -24321.2,E2 -24321.2} C_VEL
LIN {X 0,Y 143.165,Z 251.646,A -85,B 0,C 180,E1 -24327.939,E2 -24327.939} C_VEL
LIN {X 0,Y 143.145,Z 251.648,A -85,B 0,C 180,E1 -24333.439,E2 -24333.439} C_VEL
LIN {X 0,Y 143.069,Z 251.654,A -85,B 0,C 180,E1 -24339.688,E2 -24339.688} C_VEL
LIN {X 0,Y 143.055,Z 251.651,A -85,B 0,C 180,E1 -24343.456,E2 -24343.456} C_VEL
LIN {X 0,Y 143.094,Z 251.657,A -85,B 0,C 180,E1 -24349.414,E2 -24349.414} C_VEL
LIN {X 0,Y 143.046,Z 251.664,A -85,B 0,C 180,E1 -24349.968,E2 -24349.968} C_VEL
LIN {X 0,Y 144.084,Z 254.578,A -85,B 0,C 180,E1 -24350.631,E2 -24350.631} C_VEL
LIN {X 0,Y 146.454,Z 257.318,A -85,B 0,C 180,E1 -24351.761,E2 -24351.761} C_VEL
LIN {X 0,Y 148.704,Z 260.605,A -85,B 0,C 180,E1 -24352.828,E2 -24352.828} C_VEL
LIN {X 0,Y 156.053,Z 272.194,A -85,B 0,C 180,E1 -24356.037,E2 -24356.037} C_VEL
LIN {X 0,Y 162.068,Z 283.37,A -85,B 0,C 180,E1 -24358.447,E2 -24358.447} C_VEL
LIN {X 0,Y 167.272,Z 294.616,A -85,B 0,C 180,E1 -24360.423,E2 -24360.423} C_VEL
LIN {X 0,Y 167.702,Z 295.961,A -85,B 0,C 180,E1 -24360.6,E2 -24360.6} C_VEL
LIN {X 0,Y 164.527,Z 348.67,A -85,B 0,C 180,E1 -24362.672,E2 -24362.672} C_VEL
LIN {X 0,Y 163,Z 362.306,A -85,B 0,C 180,E1 -24363.694,E2 -24363.694} C_VEL
LIN {X 0,Y 161.018,Z 375.068,A -85,B 0,C 180,E1 -24365.167,E2 -24365.167} C_VEL
LIN {X 0,Y 158.504,Z 387.523,A -85,B 0,C 180,E1 -24367.179,E2 -24367.179} C_VEL
LIN {X 0,Y 155.548,Z 398.692,A -85,B 0,C 180,E1 -24369.51,E2 -24369.51} C_VEL
LIN {X 0,Y 152.965,Z 407.705,A -85,B 0,C 180,E1 -24371.94,E2 -24371.94} C_VEL
LIN {X 0,Y 149.945,Z 416.979,A -85,B 0,C 180,E1 -24375.068,E2 -24375.068} C_VEL
LIN {X 0,Y 147.04,Z 425.946,A -85,B 0,C 180,E1 -24378.984,E2 -24378.984} C_VEL
LIN {X 0,Y 144.52,Z 433.201,A -85,B 0,C 180,E1 -24383.023,E2 -24383.023} C_VEL
LIN {X 0,Y 142.869,Z 438.978,A -85,B 0,C 180,E1 -24387.186,E2 -24387.186} C_VEL
LIN {X 0,Y 141.687,Z 443.542,A -85,B 0,C 180,E1 -24391.426,E2 -24391.426} C_VEL
LIN {X 0,Y 140.947,Z 447.033,A -85,B 0,C 180,E1 -24395.728,E2 -24395.728} C_VEL
LIN {X 0,Y 140.602,Z 448.789,A -85,B 0,C 180,E1 -24398.629,E2 -24398.629} C_VEL
LIN {X 0,Y 140.546,Z 450.134,A -85,B 0,C 180,E1 -24401.542,E2 -24401.542} C_VEL
LIN {X 0,Y 140.748,Z 451.083,A -85,B 0,C 180,E1 -24404.462,E2 -24404.462} C_VEL
LIN {X 0,Y 141.792,Z 451.737,A -85,B 0,C 180,E1 -24409.651,E2 -24409.651} C_VEL
LIN {X 0,Y 142.935,Z 451.421,A -85,B 0,C 180,E1 -24413.167,E2 -24413.167} C_VEL
LIN {X 0,Y 144.217,Z 450.735,A -85,B 0,C 180,E1 -24416.017,E2 -24416.017} C_VEL
LIN {X 0,Y 147.07,Z 448.607,A -85,B 0,C 180,E1 -24420.664,E2 -24420.664} C_VEL
LIN {X 0,Y 151.107,Z 444.819,A -85,B 0,C 180,E1 -24425.55,E2 -24425.55} C_VEL
LIN {X 0,Y 155.864,Z 439.708,A -85,B 0,C 180,E1 -24429.955,E2 -24429.955} C_VEL
LIN {X 0,Y 160.639,Z 433.877,A -85,B 0,C 180,E1 -24433.557,E2 -24433.557} C_VEL
LIN {X 0,Y 166.329,Z 426.027,A -85,B 0,C 180,E1 -24437.12,E2 -24437.12} C_VEL
LIN {X 0,Y 171.796,Z 417.358,A -85,B 0,C 180,E1 -24440.089,E2 -24440.089} C_VEL
LIN {X 0,Y 177.003,Z 407.771,A -85,B 0,C 180,E1 -24442.571,E2 -24442.571} C_VEL
LIN {X 0,Y 181.501,Z 398.125,A -85,B 0,C 180,E1 -24444.491,E2 -24444.491} C_VEL
LIN {X 0,Y 185.86,Z 386.627,A -85,B 0,C 180,E1 -24446.293,E2 -24446.293} C_VEL
LIN {X 0,Y 189.344,Z 375.321,A -85,B 0,C 180,E1 -24447.609,E2 -24447.609} C_VEL
LIN {X 0,Y 192.409,Z 362.116,A -85,B 0,C 180,E1 -24448.69,E2 -24448.69} C_VEL
LIN {X 0,Y 194.374,Z 349.343,A -85,B 0,C 180,E1 -24449.401,E2 -24449.401} C_VEL
LIN {X 0,Y 196.628,Z 322.015,A -85,B 0,C 180,E1 -24450.282,E2 -24450.282} C_VEL
LIN {X 0,Y 191.407,Z 312.105,A -85,B 0,C 180,E1 -24453.214,E2 -24453.214} C_VEL
LIN {X 0,Y 185.703,Z 302.569,A -85,B 0,C 180,E1 -24456.844,E2 -24456.844} C_VEL
LIN {X 0,Y 182.192,Z 297.271,A -85,B 0,C 180,E1 -24459.39,E2 -24459.39} C_VEL
LIN {X 0,Y 179.939,Z 293.977,A -85,B 0,C 180,E1 -24461.202,E2 -24461.202} C_VEL
LIN {X 0,Y 177.659,Z 290.688,A -85,B 0,C 180,E1 -24463.222,E2 -24463.222} C_VEL
LIN {X 0,Y 174.991,Z 286.951,A -85,B 0,C 180,E1 -24465.908,E2 -24465.908} C_VEL
LIN {X 0,Y 174.118,Z 285.861,A -85,B 0,C 180,E1 -24466.877,E2 -24466.877} C_VEL
LIN {X 0,Y 171.735,Z 282.687,A -85,B 0,C 180,E1 -24469.906,E2 -24469.906} C_VEL
LIN {X 0,Y 171.049,Z 281.31,A -85,B 0,C 180,E1 -24470.988,E2 -24470.988} C_VEL
LIN {X 0,Y 168.374,Z 278.475,A -85,B 0,C 180,E1 -24475.811,E2 -24475.811} C_VEL
LIN {X 0,Y 167.446,Z 275.959,A -85,B 0,C 180,E1 -24478.797,E2 -24478.797} C_VEL
LIN {X 0,Y 166.615,Z 275.627,A -85,B 0,C 180,E1 -24482.417,E2 -24482.417} C_VEL
LIN {X 0,Y 167.321,Z 276.079,A -85,B 0,C 180,E1 -24491.274,E2 -24491.274} C_VEL
LIN {X 0,Y 168.57,Z 279.27,A -85,B 0,C 180,E1 -24495.181,E2 -24495.181} C_VEL
LIN {X 0,Y 171.269,Z 281.913,A -85,B 0,C 180,E1 -24499.811,E2 -24499.811} C_VEL
LIN {X 0,Y 175.325,Z 288.276,A -85,B 0,C 180,E1 -24504.975,E2 -24504.975} C_VEL
LIN {X 0,Y 178.922,Z 294.333,A -85,B 0,C 180,E1 -24508.522,E2 -24508.522} C_VEL
LIN {X 0,Y 182.114,Z 300.198,A -85,B 0,C 180,E1 -24511.236,E2 -24511.236} C_VEL
LIN {X 0,Y 185.998,Z 307.662,A -85,B 0,C 180,E1 -24514.136,E2 -24514.136} C_VEL
LIN {X 0,Y 189.951,Z 316.155,A -85,B 0,C 180,E1 -24516.793,E2 -24516.793} C_VEL
LIN {X 0,Y 194.142,Z 326.143,A -85,B 0,C 180,E1 -24519.358,E2 -24519.358} C_VEL
LIN {X 0,Y 195.955,Z 331.201,A -85,B 0,C 180,E1 -24520.432,E2 -24520.432} C_VEL
LIN {X 0,Y 193.595,Z 360.249,A -85,B 0,C 180,E1 -24521.381,E2 -24521.381} C_VEL
LIN {X 0,Y 191.386,Z 373.578,A -85,B 0,C 180,E1 -24522.079,E2 -24522.079} C_VEL
LIN {X 0,Y 188.213,Z 386.396,A -85,B 0,C 180,E1 -24523.074,E2 -24523.074} C_VEL
LIN {X 0,Y 184.224,Z 398.185,A -85,B 0,C 180,E1 -24524.332,E2 -24524.332} C_VEL
LIN {X 0,Y 179.568,Z 409.533,A -85,B 0,C 180,E1 -24525.996,E2 -24525.996} C_VEL
LIN {X 0,Y 174.585,Z 419.788,A -85,B 0,C 180,E1 -24527.99,E2 -24527.99} C_VEL
LIN {X 0,Y 169.803,Z 428.197,A -85,B 0,C 180,E1 -24530.093,E2 -24530.093} C_VEL
LIN {X 0,Y 163.982,Z 437.334,A -85,B 0,C 180,E1 -24533.127,E2 -24533.127} C_VEL
LIN {X 0,Y 158.587,Z 444.72,A -85,B 0,C 180,E1 -24536.359,E2 -24536.359} C_VEL
LIN {X 0,Y 153.941,Z 450.672,A -85,B 0,C 180,E1 -24539.852,E2 -24539.852} C_VEL
LIN {X 0,Y 150.047,Z 455.402,A -85,B 0,C 180,E1 -24543.576,E2 -24543.576} C_VEL
LIN {X 0,Y 146.641,Z 459.045,A -85,B 0,C 180,E1 -24547.452,E2 -24547.452} C_VEL
LIN {X 0,Y 144.793,Z 460.946,A -85,B 0,C 180,E1 -24550.134,E2 -24550.134} C_VEL
LIN {X 0,Y 143.239,Z 462.394,A -85,B 0,C 180,E1 -24552.875,E2 -24552.875} C_VEL
LIN {X 0,Y 141.345,Z 464.127,A -85,B 0,C 180,E1 -24558.524,E2 -24558.524} C_VEL
LIN {X 0,Y 140.895,Z 464.379,A -85,B 0,C 180,E1 -24560.944,E2 -24560.944} C_VEL
LIN {X 0,Y 140.005,Z 464.423,A -85,B 0,C 180,E1 -24563.33,E2 -24563.33} C_VEL
LIN {X 0,Y 138.351,Z 464.089,A -85,B 0,C 180,E1 -24565.682,E2 -24565.682} C_VEL
LIN {X 0,Y 134.708,Z 462.414,A -85,B 0,C 180,E1 -24570.452,E2 -24570.452} C_VEL
LIN {X 0,Y 133.616,Z 460.619,A -85,B 0,C 180,E1 -24573.76,E2 -24573.76} C_VEL
LIN {X 0,Y 133.761,Z 458.148,A -85,B 0,C 180,E1 -24577.541,E2 -24577.541} C_VEL
LIN {X 0,Y 134.318,Z 454.139,A -85,B 0,C 180,E1 -24582.074,E2 -24582.074} C_VEL
LIN {X 0,Y 135.854,Z 447.945,A -85,B 0,C 180,E1 -24587.297,E2 -24587.297} C_VEL
LIN {X 0,Y 138.014,Z 441.169,A -85,B 0,C 180,E1 -24591.657,E2 -24591.657} C_VEL
LIN {X 0,Y 140.08,Z 434.831,A -85,B 0,C 180,E1 -24594.926,E2 -24594.926} C_VEL
LIN {X 0,Y 143.29,Z 425.927,A -85,B 0,C 180,E1 -24598.56,E2 -24598.56} C_VEL
LIN {X 0,Y 146.508,Z 415.695,A -85,B 0,C 180,E1 -24601.839,E2 -24601.839} C_VEL
LIN {X 0,Y 149.591,Z 405.561,A -85,B 0,C 180,E1 -24604.307,E2 -24604.307} C_VEL
LIN {X 0,Y 152.511,Z 394.517,A -85,B 0,C 180,E1 -24606.381,E2 -24606.381} C_VEL
LIN {X 0,Y 155.185,Z 382.289,A -85,B 0,C 180,E1 -24608.09,E2 -24608.09} C_VEL
LIN {X 0,Y 157.209,Z 370.071,A -85,B 0,C 180,E1 -24609.295,E2 -24609.295} C_VEL
LIN {X 0,Y 158.616,Z 356.285,A -85,B 0,C 180,E1 -24610.157,E2 -24610.157} C_VEL
LIN {X 0,Y 160.749,Z 319.162,A -85,B 0,C 180,E1 -24611.659,E2 -24611.659} C_VEL
LIN {X 0,Y 159.496,Z 299.831,A -85,B 0,C 180,E1 -24613.072,E2 -24613.072} C_VEL
LIN {X 0,Y 154.959,Z 287.258,A -85,B 0,C 180,E1 -24615.131,E2 -24615.131} C_VEL
LIN {X 0,Y 150.7,Z 277.42,A -85,B 0,C 180,E1 -24617.11,E2 -24617.11} C_VEL
LIN {X 0,Y 146.197,Z 268.432,A -85,B 0,C 180,E1 -24619.309,E2 -24619.309} C_VEL
LIN {X 0,Y 144.29,Z 265.293,A -85,B 0,C 180,E1 -24620.262,E2 -24620.262} C_VEL
LIN {X 0,Y 141.666,Z 261.495,A -85,B 0,C 180,E1 -24621.602,E2 -24621.602} C_VEL
LIN {X 0,Y 139.477,Z 258.156,A -85,B 0,C 180,E1 -24622.796,E2 -24622.796} C_VEL
LIN {X 0,Y 138.54,Z 257.091,A -85,B 0,C 180,E1 -24623.298,E2 -24623.298} C_VEL
LIN {X 0,Y 136.72,Z 254.771,A -85,B 0,C 180,E1 -24624.33,E2 -24624.33} C_VEL
LIN {X 0,Y 136.046,Z 252.541,A -85,B 0,C 180,E1 -24624.921,E2 -24624.921} C_VEL
LIN {X 0,Y 136.077,Z 252.536,A -85,B 0,C 180,E1 -24631.381,E2 -24631.381} C_VEL
LIN {X 0,Y 136.253,Z 252.512,A -85,B 0,C 180,E1 -24638.835,E2 -24638.835} C_VEL
LIN {X 0,Y 136.24,Z 252.51,A -85,B 0,C 180,E1 -24645.053,E2 -24645.053} C_VEL
LIN {X 0,Y 136.4,Z 252.489,A -85,B 0,C 180,E1 -24648.175,E2 -24648.175} C_VEL
LIN {X 0,Y 136.52,Z 252.474,A -85,B 0,C 180,E1 -24651.116,E2 -24651.116} C_VEL
LIN {X 0,Y 137.09,Z 252.37,A -85,B 0,C 180,E1 -24660,E2 -24660} C_VEL
LIN {X 0,Y 136.517,Z 252.477,A -85,B 0,C 180,E1 -24668.885,E2 -24668.885} C_VEL
LIN {X 0,Y 136.387,Z 252.466,A -85,B 0,C 180,E1 -24671.895,E2 -24671.895} C_VEL
LIN {X 0,Y 136.137,Z 252.512,A -85,B 0,C 180,E1 -24678.044,E2 -24678.044} C_VEL
LIN {X 0,Y 136.123,Z 252.525,A -85,B 0,C 180,E1 -24681.698,E2 -24681.698} C_VEL
LIN {X 0,Y 136.076,Z 252.526,A -85,B 0,C 180,E1 -24688.619,E2 -24688.619} C_VEL
LIN {X 0,Y 136.058,Z 252.528,A -85,B 0,C 180,E1 -24694.625,E2 -24694.625} C_VEL
LIN {X 0,Y 136.041,Z 252.529,A -85,B 0,C 180,E1 -24699.218,E2 -24699.218} C_VEL
LIN {X 0,Y 135.994,Z 252.526,A -85,B 0,C 180,E1 -24703.67,E2 -24703.67} C_VEL
LIN {X 0,Y 136.01,Z 252.606,A -85,B 0,C 180,E1 -24706.877,E2 -24706.877} C_VEL
LIN {X 0,Y 136.944,Z 255.258,A -85,B 0,C 180,E1 -24707.539,E2 -24707.539} C_VEL
LIN {X 0,Y 139.404,Z 258.038,A -85,B 0,C 180,E1 -24708.887,E2 -24708.887} C_VEL
LIN {X 0,Y 141.391,Z 261.22,A -85,B 0,C 180,E1 -24709.986,E2 -24709.986} C_VEL
LIN {X 0,Y 142.836,Z 263.062,A -85,B 0,C 180,E1 -24710.72,E2 -24710.72} C_VEL
LIN {X 0,Y 148.081,Z 271.025,A -85,B 0,C 180,E1 -24713.285,E2 -24713.285} C_VEL
LIN {X 0,Y 153.283,Z 279.825,A -85,B 0,C 180,E1 -24715.619,E2 -24715.619} C_VEL
LIN {X 0,Y 159.477,Z 292.071,A -85,B 0,C 180,E1 -24718.209,E2 -24718.209} C_VEL
LIN {X 0,Y 161.878,Z 298.045,A -85,B 0,C 180,E1 -24719.207,E2 -24719.207} C_VEL
LIN {X 0,Y 158.727,Z 348.407,A -85,B 0,C 180,E1 -24721.224,E2 -24721.224} C_VEL
LIN {X 0,Y 157.081,Z 362.258,A -85,B 0,C 180,E1 -24722.26,E2 -24722.26} C_VEL
LIN {X 0,Y 155.028,Z 375.138,A -85,B 0,C 180,E1 -24723.776,E2 -24723.776} C_VEL
LIN {X 0,Y 152.407,Z 387.64,A -85,B 0,C 180,E1 -24725.85,E2 -24725.85} C_VEL
LIN {X 0,Y 149.308,Z 398.847,A -85,B 0,C 180,E1 -24728.25,E2 -24728.25} C_VEL
LIN {X 0,Y 146.196,Z 408.918,A -85,B 0,C 180,E1 -24731.073,E2 -24731.073} C_VEL
LIN {X 0,Y 143.134,Z 418.007,A -85,B 0,C 180,E1 -24734.34,E2 -24734.34} C_VEL
LIN {X 0,Y 140.073,Z 426.862,A -85,B 0,C 180,E1 -24738.429,E2 -24738.429} C_VEL
LIN {X 0,Y 137.473,Z 433.999,A -85,B 0,C 180,E1 -24742.663,E2 -24742.663} C_VEL
LIN {X 0,Y 135.78,Z 439.661,A -85,B 0,C 180,E1 -24747.039,E2 -24747.039} C_VEL
LIN {X 0,Y 134.575,Z 444.142,A -85,B 0,C 180,E1 -24751.502,E2 -24751.502} C_VEL
LIN {X 0,Y 133.8,Z 447.564,A -85,B 0,C 180,E1 -24756.035,E2 -24756.035} C_VEL
LIN {X 0,Y 133.483,Z 449.28,A -85,B 0,C 180,E1 -24759.093,E2 -24759.093} C_VEL
LIN {X 0,Y 133.475,Z 450.59,A -85,B 0,C 180,E1 -24762.163,E2 -24762.163} C_VEL
LIN {X 0,Y 133.763,Z 451.498,A -85,B 0,C 180,E1 -24765.235,E2 -24765.235} C_VEL
LIN {X 0,Y 134.83,Z 452.071,A -85,B 0,C 180,E1 -24770.239,E2 -24770.239} C_VEL
LIN {X 0,Y 136.248,Z 451.703,A -85,B 0,C 180,E1 -24774.376,E2 -24774.376} C_VEL
LIN {X 0,Y 137.679,Z 450.965,A -85,B 0,C 180,E1 -24777.353,E2 -24777.353} C_VEL
LIN {X 0,Y 140.495,Z 449.015,A -85,B 0,C 180,E1 -24781.744,E2 -24781.744} C_VEL
LIN {X 0,Y 143.91,Z 446.115,A -85,B 0,C 180,E1 -24785.878,E2 -24785.878} C_VEL
LIN {X 0,Y 148.048,Z 442.097,A -85,B 0,C 180,E1 -24789.858,E2 -24789.858} C_VEL
LIN {X 0,Y 153.69,Z 435.833,A -85,B 0,C 180,E1 -24794.217,E2 -24794.217} C_VEL
LIN {X 0,Y 159.15,Z 428.954,A -85,B 0,C 180,E1 -24797.705,E2 -24797.705} C_VEL
LIN {X 0,Y 164.052,Z 421.881,A -85,B 0,C 180,E1 -24800.455,E2 -24800.455} C_VEL
LIN {X 0,Y 169.373,Z 413.306,A -85,B 0,C 180,E1 -24803.012,E2 -24803.012} C_VEL
LIN {X 0,Y 174.618,Z 403.313,A -85,B 0,C 180,E1 -24805.299,E2 -24805.299} C_VEL
LIN {X 0,Y 179.582,Z 391.936,A -85,B 0,C 180,E1 -24807.288,E2 -24807.288} C_VEL
LIN {X 0,Y 183.67,Z 380.017,A -85,B 0,C 180,E1 -24808.887,E2 -24808.887} C_VEL
LIN {X 0,Y 187.055,Z 367.754,A -85,B 0,C 180,E1 -24810.012,E2 -24810.012} C_VEL
LIN {X 0,Y 189.567,Z 354.481,A -85,B 0,C 180,E1 -24810.897,E2 -24810.897} C_VEL
LIN {X 0,Y 191.093,Z 341.157,A -85,B 0,C 180,E1 -24811.404,E2 -24811.404} C_VEL
LIN {X 0,Y 192.334,Z 325.055,A -85,B 0,C 180,E1 -24811.917,E2 -24811.917} C_VEL
LIN {X 0,Y 187.644,Z 316.143,A -85,B 0,C 180,E1 -24814.769,E2 -24814.769} C_VEL
LIN {X 0,Y 182.855,Z 307.914,A -85,B 0,C 180,E1 -24818.066,E2 -24818.066} C_VEL
LIN {X 0,Y 178.557,Z 301.115,A -85,B 0,C 180,E1 -24821.498,E2 -24821.498} C_VEL
LIN {X 0,Y 175.748,Z 297.055,A -85,B 0,C 180,E1 -24824.079,E2 -24824.079} C_VEL
LIN {X 0,Y 172.714,Z 292.64,A -85,B 0,C 180,E1 -24827.396,E2 -24827.396} C_VEL
LIN {X 0,Y 170.383,Z 289.442,A -85,B 0,C 180,E1 -24830.503,E2 -24830.503} C_VEL
LIN {X 0,Y 169.612,Z 288.021,A -85,B 0,C 180,E1 -24831.767,E2 -24831.767} C_VEL
LIN {X 0,Y 167.128,Z 285.057,A -85,B 0,C 180,E1 -24836.699,E2 -24836.699} C_VEL
LIN {X 0,Y 166.468,Z 282.957,A -85,B 0,C 180,E1 -24839.128,E2 -24839.128} C_VEL
LIN {X 0,Y 165.521,Z 282.775,A -85,B 0,C 180,E1 -24844.871,E2 -24844.871} C_VEL
LIN {X 0,Y 166.34,Z 283.178,A -85,B 0,C 180,E1 -24850.96,E2 -24850.96} C_VEL
LIN {X 0,Y 167.728,Z 286.516,A -85,B 0,C 180,E1 -24855.318,E2 -24855.318} C_VEL
LIN {X 0,Y 169.929,Z 288.704,A -85,B 0,C 180,E1 -24859.201,E2 -24859.201} C_VEL
LIN {X 0,Y 173.566,Z 294.659,A -85,B 0,C 180,E1 -24864.124,E2 -24864.124} C_VEL
LIN {X 0,Y 176.84,Z 300.469,A -85,B 0,C 180,E1 -24867.577,E2 -24867.577} C_VEL
LIN {X 0,Y 179.754,Z 306.093,A -85,B 0,C 180,E1 -24870.223,E2 -24870.223} C_VEL
LIN {X 0,Y 183.29,Z 313.236,A -85,B 0,C 180,E1 -24873.053,E2 -24873.053} C_VEL
LIN {X 0,Y 187.134,Z 321.895,A -85,B 0,C 180,E1 -24875.812,E2 -24875.812} C_VEL
LIN {X 0,Y 191.045,Z 331.843,A -85,B 0,C 180,E1 -24878.375,E2 -24878.375} C_VEL
LIN {X 0,Y 191.718,Z 333.772,A -85,B 0,C 180,E1 -24878.803,E2 -24878.803} C_VEL
LIN {X 0,Y 189.394,Z 360.411,A -85,B 0,C 180,E1 -24879.669,E2 -24879.669} C_VEL
LIN {X 0,Y 187.091,Z 373.74,A -85,B 0,C 180,E1 -24880.376,E2 -24880.376} C_VEL
LIN {X 0,Y 183.791,Z 386.474,A -85,B 0,C 180,E1 -24881.371,E2 -24881.371} C_VEL
LIN {X 0,Y 179.365,Z 398.966,A -85,B 0,C 180,E1 -24882.72,E2 -24882.72} C_VEL
LIN {X 0,Y 174.559,Z 410.111,A -85,B 0,C 180,E1 -24884.386,E2 -24884.386} C_VEL
LIN {X 0,Y 169.962,Z 419.145,A -85,B 0,C 180,E1 -24886.161,E2 -24886.161} C_VEL
LIN {X 0,Y 165.479,Z 426.718,A -85,B 0,C 180,E1 -24888.016,E2 -24888.016} C_VEL
LIN {X 0,Y 160.321,Z 434.689,A -85,B 0,C 180,E1 -24890.531,E2 -24890.531} C_VEL
LIN {X 0,Y 154.558,Z 442.537,A -85,B 0,C 180,E1 -24893.761,E2 -24893.761} C_VEL
LIN {X 0,Y 149.352,Z 448.834,A -85,B 0,C 180,E1 -24897.236,E2 -24897.236} C_VEL
LIN {X 0,Y 144.986,Z 453.878,A -85,B 0,C 180,E1 -24901.002,E2 -24901.002} C_VEL
LIN {X 0,Y 141.187,Z 457.817,A -85,B 0,C 180,E1 -24904.966,E2 -24904.966} C_VEL
LIN {X 0,Y 138.107,Z 460.753,A -85,B 0,C 180,E1 -24909.128,E2 -24909.128} C_VEL
LIN {X 0,Y 135.243,Z 463.19,A -85,B 0,C 180,E1 -24914.936,E2 -24914.936} C_VEL
LIN {X 0,Y 133.812,Z 464.102,A -85,B 0,C 180,E1 -24920.93,E2 -24920.93} C_VEL
LIN {X 0,Y 133.61,Z 463.944,A -85,B 0,C 180,E1 -24923.956,E2 -24923.956} C_VEL
LIN {X 0,Y 133.652,Z 463.25,A -85,B 0,C 180,E1 -24927.576,E2 -24927.576} C_VEL
LIN {X 0,Y 133.814,Z 462.459,A -85,B 0,C 180,E1 -24929.994,E2 -24929.994} C_VEL
LIN {X 0,Y 133.616,Z 460.619,A -85,B 0,C 180,E1 -24933.76,E2 -24933.76} C_VEL
LIN {X 0,Y 132.966,Z 459.096,A -85,B 0,C 180,E1 -24936.187,E2 -24936.187} C_VEL
LIN {X 0,Y 130.396,Z 455.958,A -85,B 0,C 180,E1 -24940.134,E2 -24940.134} C_VEL
LIN {X 0,Y 128.273,Z 452.142,A -85,B 0,C 180,E1 -24944.116,E2 -24944.116} C_VEL
LIN {X 0,Y 128.349,Z 449.459,A -85,B 0,C 180,E1 -24946.493,E2 -24946.493} C_VEL
LIN {X 0,Y 130.588,Z 442.901,A -85,B 0,C 180,E1 -24951.293,E2 -24951.293} C_VEL
LIN {X 0,Y 133.299,Z 434.844,A -85,B 0,C 180,E1 -24955.808,E2 -24955.808} C_VEL
LIN {X 0,Y 136.387,Z 426.785,A -85,B 0,C 180,E1 -24959.3,E2 -24959.3} C_VEL
LIN {X 0,Y 139.777,Z 416.83,A -85,B 0,C 180,E1 -24962.708,E2 -24962.708} C_VEL
LIN {X 0,Y 142.493,Z 408.369,A -85,B 0,C 180,E1 -24964.975,E2 -24964.975} C_VEL
LIN {X 0,Y 145.508,Z 398.149,A -85,B 0,C 180,E1 -24967.128,E2 -24967.128} C_VEL
LIN {X 0,Y 148.487,Z 386.1,A -85,B 0,C 180,E1 -24969.046,E2 -24969.046} C_VEL
LIN {X 0,Y 150.817,Z 373.406,A -85,B 0,C 180,E1 -24970.491,E2 -24970.491} C_VEL
LIN {X 0,Y 152.615,Z 359.806,A -85,B 0,C 180,E1 -24971.488,E2 -24971.488} C_VEL
LIN {X 0,Y 155.04,Z 319.438,A -85,B 0,C 180,E1 -24973.217,E2 -24973.217} C_VEL
LIN {X 0,Y 153.964,Z 302.059,A -85,B 0,C 180,E1 -24974.555,E2 -24974.555} C_VEL
LIN {X 0,Y 150.057,Z 290.914,A -85,B 0,C 180,E1 -24976.478,E2 -24976.478} C_VEL
LIN {X 0,Y 146.227,Z 281.793,A -85,B 0,C 180,E1 -24978.405,E2 -24978.405} C_VEL
LIN {X 0,Y 141.068,Z 271.303,A -85,B 0,C 180,E1 -24981.147,E2 -24981.147} C_VEL
LIN {X 0,Y 137.883,Z 266.721,A -85,B 0,C 180,E1 -24982.866,E2 -24982.866} C_VEL
LIN {X 0,Y 135.184,Z 262.821,A -85,B 0,C 180,E1 -24984.435,E2 -24984.435} C_VEL
LIN {X 0,Y 132.978,Z 259.722,A -85,B 0,C 180,E1 -24985.798,E2 -24985.798} C_VEL
LIN {X 0,Y 132.265,Z 258.552,A -85,B 0,C 180,E1 -24986.27,E2 -24986.27} C_VEL
LIN {X 0,Y 130.091,Z 256.451,A -85,B 0,C 180,E1 -24987.645,E2 -24987.645} C_VEL
LIN {X 0,Y 129.123,Z 254.178,A -85,B 0,C 180,E1 -24988.408,E2 -24988.408} C_VEL
LIN {X 0,Y 128.98,Z 253.419,A -85,B 0,C 180,E1 -24988.597,E2 -24988.597} C_VEL
LIN {X 0,Y 129.013,Z 253.412,A -85,B 0,C 180,E1 -24994.164,E2 -24994.164} C_VEL
LIN {X 0,Y 129.105,Z 253.398,A -85,B 0,C 180,E1 -24997.702,E2 -24997.702} C_VEL
LIN {X 0,Y 129.149,Z 253.393,A -85,B 0,C 180,E1 -25000.943,E2 -25000.943} C_VEL
LIN {X 0,Y 129.325,Z 253.368,A -85,B 0,C 180,E1 -25007.956,E2 -25007.956} C_VEL
LIN {X 0,Y 129.444,Z 253.358,A -85,B 0,C 180,E1 -25010.626,E2 -25010.626} C_VEL
LIN {X 0,Y 130.045,Z 253.246,A -85,B 0,C 180,E1 -25020,E2 -25020} C_VEL
LIN {X 0,Y 129.441,Z 253.357,A -85,B 0,C 180,E1 -25029.375,E2 -25029.375} C_VEL
LIN {X 0,Y 129.271,Z 253.343,A -85,B 0,C 180,E1 -25032.561,E2 -25032.561} C_VEL
LIN {X 0,Y 129.056,Z 253.403,A -85,B 0,C 180,E1 -25039.071,E2 -25039.071} C_VEL
LIN {X 0,Y 129.021,Z 253.405,A -85,B 0,C 180,E1 -25042.415,E2 -25042.415} C_VEL
LIN {X 0,Y 128.988,Z 253.417,A -85,B 0,C 180,E1 -25045.842,E2 -25045.842} C_VEL
LIN {X 0,Y 128.996,Z 253.407,A -85,B 0,C 180,E1 -25049.363,E2 -25049.363} C_VEL
LIN {X 0,Y 128.973,Z 253.412,A -85,B 0,C 180,E1 -25055.195,E2 -25055.195} C_VEL
LIN {X 0,Y 128.965,Z 253.415,A -85,B 0,C 180,E1 -25060.841,E2 -25060.841} C_VEL
LIN {X 0,Y 128.951,Z 253.408,A -85,B 0,C 180,E1 -25063.144,E2 -25063.144} C_VEL
LIN {X 0,Y 129.864,Z 256.1,A -85,B 0,C 180,E1 -25063.924,E2 -25063.924} C_VEL
LIN {X 0,Y 131.851,Z 258.314,A -85,B 0,C 180,E1 -25065.218,E2 -25065.218} C_VEL
LIN {X 0,Y 132.61,Z 259.036,A -85,B 0,C 180,E1 -25065.682,E2 -25065.682} C_VEL
LIN {X 0,Y 134.805,Z 262.424,A -85,B 0,C 180,E1 -25067.076,E2 -25067.076} C_VEL
LIN {X 0,Y 136.142,Z 264.182,A -85,B 0,C 180,E1 -25067.861,E2 -25067.861} C_VEL
LIN {X 0,Y 141.319,Z 271.674,A -85,B 0,C 180,E1 -25070.71,E2 -25070.71} C_VEL
LIN {X 0,Y 147.342,Z 281.583,A -85,B 0,C 180,E1 -25073.711,E2 -25073.711} C_VEL
LIN {X 0,Y 152.924,Z 292.443,A -85,B 0,C 180,E1 -25076.273,E2 -25076.273} C_VEL
LIN {X 0,Y 156.061,Z 299.449,A -85,B 0,C 180,E1 -25077.646,E2 -25077.646} C_VEL
LIN {X 0,Y 152.919,Z 349.255,A -85,B 0,C 180,E1 -25079.737,E2 -25079.737} C_VEL
LIN {X 0,Y 151.212,Z 362.928,A -85,B 0,C 180,E1 -25080.799,E2 -25080.799} C_VEL
LIN {X 0,Y 149.134,Z 375.196,A -85,B 0,C 180,E1 -25082.275,E2 -25082.275} C_VEL
LIN {X 0,Y 146.798,Z 386.179,A -85,B 0,C 180,E1 -25084.105,E2 -25084.105} C_VEL
LIN {X 0,Y 143.526,Z 397.713,A -85,B 0,C 180,E1 -25086.564,E2 -25086.564} C_VEL
LIN {X 0,Y 140.269,Z 408.074,A -85,B 0,C 180,E1 -25089.476,E2 -25089.476} C_VEL
LIN {X 0,Y 136.911,Z 417.416,A -85,B 0,C 180,E1 -25092.84,E2 -25092.84} C_VEL
LIN {X 0,Y 133.636,Z 426.421,A -85,B 0,C 180,E1 -25097.092,E2 -25097.092} C_VEL
LIN {X 0,Y 130.823,Z 433.706,A -85,B 0,C 180,E1 -25101.511,E2 -25101.511} C_VEL
LIN {X 0,Y 129.191,Z 438.615,A -85,B 0,C 180,E1 -25105.326,E2 -25105.326} C_VEL
LIN {X 0,Y 127.742,Z 443.4,A -85,B 0,C 180,E1 -25110.006,E2 -25110.006} C_VEL
LIN {X 0,Y 126.931,Z 447.03,A -85,B 0,C 180,E1 -25114.696,E2 -25114.696} C_VEL
LIN {X 0,Y 126.36,Z 449.773,A -85,B 0,C 180,E1 -25119.61,E2 -25119.61} C_VEL
LIN {X 0,Y 126.41,Z 451.047,A -85,B 0,C 180,E1 -25122.854,E2 -25122.854} C_VEL
LIN {X 0,Y 126.78,Z 451.892,A -85,B 0,C 180,E1 -25126.096,E2 -25126.096} C_VEL
LIN {X 0,Y 127.873,Z 452.402,A -85,B 0,C 180,E1 -25130.878,E2 -25130.878} C_VEL
LIN {X 0,Y 129.633,Z 451.985,A -85,B 0,C 180,E1 -25135.707,E2 -25135.707} C_VEL
LIN {X 0,Y 131.234,Z 451.177,A -85,B 0,C 180,E1 -25138.818,E2 -25138.818} C_VEL
LIN {X 0,Y 133.956,Z 449.429,A -85,B 0,C 180,E1 -25142.918,E2 -25142.918} C_VEL
LIN {X 0,Y 138.036,Z 446.189,A -85,B 0,C 180,E1 -25147.662,E2 -25147.662} C_VEL
LIN {X 0,Y 142.416,Z 442.177,A -85,B 0,C 180,E1 -25151.669,E2 -25151.669} C_VEL
LIN {X 0,Y 148.5,Z 435.726,A -85,B 0,C 180,E1 -25156.199,E2 -25156.199} C_VEL
LIN {X 0,Y 154.334,Z 428.749,A -85,B 0,C 180,E1 -25159.709,E2 -25159.709} C_VEL
LIN {X 0,Y 159.521,Z 421.562,A -85,B 0,C 180,E1 -25162.469,E2 -25162.469} C_VEL
LIN {X 0,Y 165.087,Z 412.795,A -85,B 0,C 180,E1 -25165.035,E2 -25165.035} C_VEL
LIN {X 0,Y 170.276,Z 403.219,A -85,B 0,C 180,E1 -25167.195,E2 -25167.195} C_VEL
LIN {X 0,Y 175.136,Z 392.48,A -85,B 0,C 180,E1 -25169.064,E2 -25169.064} C_VEL
LIN {X 0,Y 179.387,Z 380.647,A -85,B 0,C 180,E1 -25170.656,E2 -25170.656} C_VEL
LIN {X 0,Y 182.927,Z 368.273,A -85,B 0,C 180,E1 -25171.792,E2 -25171.792} C_VEL
LIN {X 0,Y 185.534,Z 355.142,A -85,B 0,C 180,E1 -25172.66,E2 -25172.66} C_VEL
LIN {X 0,Y 187.112,Z 341.939,A -85,B 0,C 180,E1 -25173.176,E2 -25173.176} C_VEL
LIN {X 0,Y 188.229,Z 328.294,A -85,B 0,C 180,E1 -25173.6,E2 -25173.6} C_VEL
LIN {X 0,Y 183.886,Z 319.926,A -85,B 0,C 180,E1 -25176.489,E2 -25176.489} C_VEL
LIN {X 0,Y 179.429,Z 312.108,A -85,B 0,C 180,E1 -25179.863,E2 -25179.863} C_VEL
LIN {X 0,Y 175.909,Z 306.497,A -85,B 0,C 180,E1 -25182.938,E2 -25182.938} C_VEL
LIN {X 0,Y 173.931,Z 303.478,A -85,B 0,C 180,E1 -25184.901,E2 -25184.901} C_VEL
LIN {X 0,Y 171.138,Z 299.218,A -85,B 0,C 180,E1 -25188.151,E2 -25188.151} C_VEL
LIN {X 0,Y 168.892,Z 295.888,A -85,B 0,C 180,E1 -25191.374,E2 -25191.374} C_VEL
LIN {X 0,Y 168.277,Z 294.796,A -85,B 0,C 180,E1 -25192.445,E2 -25192.445} C_VEL
LIN {X 0,Y 165.936,Z 291.656,A -85,B 0,C 180,E1 -25197.572,E2 -25197.572} C_VEL
LIN {X 0,Y 165.487,Z 290.017,A -85,B 0,C 180,E1 -25199.463,E2 -25199.463} C_VEL
LIN {X 0,Y 164.87,Z 289.687,A -85,B 0,C 180,E1 -25202.443,E2 -25202.443} C_VEL
LIN {X 0,Y 165.318,Z 290.142,A -85,B 0,C 180,E1 -25210.409,E2 -25210.409} C_VEL
LIN {X 0,Y 166.813,Z 293.641,A -85,B 0,C 180,E1 -25215.287,E2 -25215.287} C_VEL
LIN {X 0,Y 168.67,Z 295.65,A -85,B 0,C 180,E1 -25218.694,E2 -25218.694} C_VEL
LIN {X 0,Y 171.908,Z 301.192,A -85,B 0,C 180,E1 -25223.338,E2 -25223.338} C_VEL
LIN {X 0,Y 174.841,Z 306.681,A -85,B 0,C 180,E1 -25226.644,E2 -25226.644} C_VEL
LIN {X 0,Y 177.922,Z 312.852,A -85,B 0,C 180,E1 -25229.599,E2 -25229.599} C_VEL
LIN {X 0,Y 181.973,Z 321.729,A -85,B 0,C 180,E1 -25232.978,E2 -25232.978} C_VEL
LIN {X 0,Y 186.394,Z 332.911,A -85,B 0,C 180,E1 -25236.244,E2 -25236.244} C_VEL
LIN {X 0,Y 187.601,Z 336.326,A -85,B 0,C 180,E1 -25237.081,E2 -25237.081} C_VEL
LIN {X 0,Y 185.447,Z 360.048,A -85,B 0,C 180,E1 -25237.86,E2 -25237.86} C_VEL
LIN {X 0,Y 183.137,Z 373.086,A -85,B 0,C 180,E1 -25238.542,E2 -25238.542} C_VEL
LIN {X 0,Y 179.858,Z 385.549,A -85,B 0,C 180,E1 -25239.49,E2 -25239.49} C_VEL
LIN {X 0,Y 175.291,Z 398.171,A -85,B 0,C 180,E1 -25240.82,E2 -25240.82} C_VEL
LIN {X 0,Y 170.294,Z 409.403,A -85,B 0,C 180,E1 -25242.464,E2 -25242.464} C_VEL
LIN {X 0,Y 164.932,Z 419.545,A -85,B 0,C 180,E1 -25244.459,E2 -25244.459} C_VEL
LIN {X 0,Y 160.283,Z 427.016,A -85,B 0,C 180,E1 -25246.322,E2 -25246.322} C_VEL
LIN {X 0,Y 154.92,Z 434.883,A -85,B 0,C 180,E1 -25248.866,E2 -25248.866} C_VEL
LIN {X 0,Y 148.88,Z 442.603,A -85,B 0,C 180,E1 -25252.142,E2 -25252.142} C_VEL
LIN {X 0,Y 143.427,Z 448.824,A -85,B 0,C 180,E1 -25255.699,E2 -25255.699} C_VEL
LIN {X 0,Y 138.787,Z 453.799,A -85,B 0,C 180,E1 -25259.574,E2 -25259.574} C_VEL
LIN {X 0,Y 134.775,Z 457.673,A -85,B 0,C 180,E1 -25263.686,E2 -25263.686} C_VEL
LIN {X 0,Y 131.473,Z 460.549,A -85,B 0,C 180,E1 -25268.022,E2 -25268.022} C_VEL
LIN {X 0,Y 129.673,Z 461.929,A -85,B 0,C 180,E1 -25271.019,E2 -25271.019} C_VEL
LIN {X 0,Y 127.393,Z 463.551,A -85,B 0,C 180,E1 -25277.247,E2 -25277.247} C_VEL
LIN {X 0,Y 126.776,Z 463.764,A -85,B 0,C 180,E1 -25280.422,E2 -25280.422} C_VEL
LIN {X 0,Y 126.537,Z 463.574,A -85,B 0,C 180,E1 -25283.617,E2 -25283.617} C_VEL
LIN {X 0,Y 126.578,Z 462.694,A -85,B 0,C 180,E1 -25288.044,E2 -25288.044} C_VEL
LIN {X 0,Y 126.715,Z 462.035,A -85,B 0,C 180,E1 -25289.994,E2 -25289.994} C_VEL
LIN {X 0,Y 126.536,Z 460.3,A -85,B 0,C 180,E1 -25293.699,E2 -25293.699} C_VEL
LIN {X 0,Y 126.693,Z 457.625,A -85,B 0,C 180,E1 -25297.965,E2 -25297.965} C_VEL
LIN {X 0,Y 127.342,Z 453.552,A -85,B 0,C 180,E1 -25302.746,E2 -25302.746} C_VEL
LIN {X 0,Y 128.349,Z 449.459,A -85,B 0,C 180,E1 -25306.493,E2 -25306.493} C_VEL
LIN {X 0,Y 128.577,Z 446.597,A -85,B 0,C 180,E1 -25308.805,E2 -25308.805} C_VEL
LIN {X 0,Y 127.446,Z 441.483,A -85,B 0,C 180,E1 -25312.598,E2 -25312.598} C_VEL
LIN {X 0,Y 126.794,Z 435.752,A -85,B 0,C 180,E1 -25316.249,E2 -25316.249} C_VEL
LIN {X 0,Y 127.73,Z 431.92,A -85,B 0,C 180,E1 -25318.233,E2 -25318.233} C_VEL
LIN {X 0,Y 130.886,Z 424.015,A -85,B 0,C 180,E1 -25321.559,E2 -25321.559} C_VEL
LIN {X 0,Y 134.128,Z 414.579,A -85,B 0,C 180,E1 -25324.727,E2 -25324.727} C_VEL
LIN {X 0,Y 138.102,Z 402.933,A -85,B 0,C 180,E1 -25327.627,E2 -25327.627} C_VEL
LIN {X 0,Y 140.825,Z 393.186,A -85,B 0,C 180,E1 -25329.505,E2 -25329.505} C_VEL
LIN {X 0,Y 143.725,Z 380.74,A -85,B 0,C 180,E1 -25331.298,E2 -25331.298} C_VEL
LIN {X 0,Y 146.008,Z 367.355,A -85,B 0,C 180,E1 -25332.603,E2 -25332.603} C_VEL
LIN {X 0,Y 147.308,Z 354.982,A -85,B 0,C 180,E1 -25333.373,E2 -25333.373} C_VEL
LIN {X 0,Y 149.468,Z 319.692,A -85,B 0,C 180,E1 -25334.882,E2 -25334.882} C_VEL
LIN {X 0,Y 148.605,Z 304.287,A -85,B 0,C 180,E1 -25336.121,E2 -25336.121} C_VEL
LIN {X 0,Y 143.85,Z 290.906,A -85,B 0,C 180,E1 -25338.676,E2 -25338.676} C_VEL
LIN {X 0,Y 138.496,Z 278.934,A -85,B 0,C 180,E1 -25341.681,E2 -25341.681} C_VEL
LIN {X 0,Y 135.791,Z 274.288,A -85,B 0,C 180,E1 -25343.243,E2 -25343.243} C_VEL
LIN {X 0,Y 131.383,Z 267.876,A -85,B 0,C 180,E1 -25345.944,E2 -25345.944} C_VEL
LIN {X 0,Y 128.865,Z 264.229,A -85,B 0,C 180,E1 -25347.646,E2 -25347.646} C_VEL
LIN {X 0,Y 126.62,Z 261.559,A -85,B 0,C 180,E1 -25349.224,E2 -25349.224} C_VEL
LIN {X 0,Y 125.562,Z 259.604,A -85,B 0,C 180,E1 -25350.078,E2 -25350.078} C_VEL
LIN {X 0,Y 123.257,Z 257.638,A -85,B 0,C 180,E1 -25351.816,E2 -25351.816} C_VEL
LIN {X 0,Y 122.158,Z 255.485,A -85,B 0,C 180,E1 -25352.828,E2 -25352.828} C_VEL
LIN {X 0,Y 121.919,Z 254.294,A -85,B 0,C 180,E1 -25353.234,E2 -25353.234} C_VEL
LIN {X 0,Y 122.022,Z 254.28,A -85,B 0,C 180,E1 -25357.122,E2 -25357.122} C_VEL
LIN {X 0,Y 122.09,Z 254.276,A -85,B 0,C 180,E1 -25363.273,E2 -25363.273} C_VEL
LIN {X 0,Y 122.372,Z 254.241,A -85,B 0,C 180,E1 -25370.079,E2 -25370.079} C_VEL
LIN {X 0,Y 122.563,Z 254.214,A -85,B 0,C 180,E1 -25376.713,E2 -25376.713} C_VEL
LIN {X 0,Y 122.998,Z 254.121,A -85,B 0,C 180,E1 -25380,E2 -25380} C_VEL
LIN {X 0,Y 122.358,Z 254.231,A -85,B 0,C 180,E1 -25387.066,E2 -25387.066} C_VEL
LIN {X 0,Y 122.261,Z 254.216,A -85,B 0,C 180,E1 -25392.308,E2 -25392.308} C_VEL
LIN {X 0,Y 122.032,Z 254.247,A -85,B 0,C 180,E1 -25396.736,E2 -25396.736} C_VEL
LIN {X 0,Y 121.964,Z 254.282,A -85,B 0,C 180,E1 -25402.813,E2 -25402.813} C_VEL
LIN {X 0,Y 121.911,Z 254.295,A -85,B 0,C 180,E1 -25407.464,E2 -25407.464} C_VEL
LIN {X 0,Y 121.887,Z 254.303,A -85,B 0,C 180,E1 -25411.262,E2 -25411.262} C_VEL
LIN {X 0,Y 121.895,Z 254.299,A -85,B 0,C 180,E1 -25416.196,E2 -25416.196} C_VEL
LIN {X 0,Y 121.898,Z 254.448,A -85,B 0,C 180,E1 -25418.594,E2 -25418.594} C_VEL
LIN {X 0,Y 122.581,Z 256.62,A -85,B 0,C 180,E1 -25419.326,E2 -25419.326} C_VEL
LIN {X 0,Y 124.67,Z 259.058,A -85,B 0,C 180,E1 -25421.015,E2 -25421.015} C_VEL
LIN {X 0,Y 125.9,Z 260.104,A -85,B 0,C 180,E1 -25421.915,E2 -25421.915} C_VEL
LIN {X 0,Y 127.76,Z 263.206,A -85,B 0,C 180,E1 -25423.347,E2 -25423.347} C_VEL
LIN {X 0,Y 129.482,Z 265.064,A -85,B 0,C 180,E1 -25424.507,E2 -25424.507} C_VEL
LIN {X 0,Y 133.007,Z 270.26,A -85,B 0,C 180,E1 -25426.821,E2 -25426.821} C_VEL
LIN {X 0,Y 137.413,Z 276.693,A -85,B 0,C 180,E1 -25429.407,E2 -25429.407} C_VEL
LIN {X 0,Y 143.244,Z 286.587,A -85,B 0,C 180,E1 -25432.524,E2 -25432.524} C_VEL
LIN {X 0,Y 148.457,Z 297.089,A -85,B 0,C 180,E1 -25435.099,E2 -25435.099} C_VEL
LIN {X 0,Y 150.504,Z 301.75,A -85,B 0,C 180,E1 -25436.069,E2 -25436.069} C_VEL
LIN {X 0,Y 147.334,Z 349.037,A -85,B 0,C 180,E1 -25438.07,E2 -25438.07} C_VEL
LIN {X 0,Y 145.564,Z 362.802,A -85,B 0,C 180,E1 -25439.146,E2 -25439.146} C_VEL
LIN {X 0,Y 143.364,Z 375.21,A -85,B 0,C 180,E1 -25440.654,E2 -25440.654} C_VEL
LIN {X 0,Y 140.91,Z 386.269,A -85,B 0,C 180,E1 -25442.535,E2 -25442.535} C_VEL
LIN {X 0,Y 137.474,Z 397.845,A -85,B 0,C 180,E1 -25445.063,E2 -25445.063} C_VEL
LIN {X 0,Y 134.039,Z 408.239,A -85,B 0,C 180,E1 -25448.072,E2 -25448.072} C_VEL
LIN {X 0,Y 130.798,Z 416.764,A -85,B 0,C 180,E1 -25451.201,E2 -25451.201} C_VEL
LIN {X 0,Y 127.803,Z 424.6,A -85,B 0,C 180,E1 -25454.866,E2 -25454.866} C_VEL
LIN {X 0,Y 124.7,Z 432.27,A -85,B 0,C 180,E1 -25459.453,E2 -25459.453} C_VEL
LIN {X 0,Y 122.113,Z 439.329,A -85,B 0,C 180,E1 -25465.054,E2 -25465.054} C_VEL
LIN {X 0,Y 120.633,Z 444.032,A -85,B 0,C 180,E1 -25470.006,E2 -25470.006} C_VEL
LIN {X 0,Y 119.845,Z 447.279,A -85,B 0,C 180,E1 -25474.491,E2 -25474.491} C_VEL
LIN {X 0,Y 119.266,Z 450.261,A -85,B 0,C 180,E1 -25480.188,E2 -25480.188} C_VEL
LIN {X 0,Y 119.363,Z 451.496,A -85,B 0,C 180,E1 -25483.627,E2 -25483.627} C_VEL
LIN {X 0,Y 119.841,Z 452.276,A -85,B 0,C 180,E1 -25487.056,E2 -25487.056} C_VEL
LIN {X 0,Y 120.919,Z 452.729,A -85,B 0,C 180,E1 -25491.572,E2 -25491.572} C_VEL
LIN {X 0,Y 123.091,Z 452.252,A -85,B 0,C 180,E1 -25497.183,E2 -25497.183} C_VEL
LIN {X 0,Y 124.88,Z 451.39,A -85,B 0,C 180,E1 -25500.435,E2 -25500.435} C_VEL
LIN {X 0,Y 127.498,Z 449.831,A -85,B 0,C 180,E1 -25504.224,E2 -25504.224} C_VEL
LIN {X 0,Y 132.311,Z 446.253,A -85,B 0,C 180,E1 -25509.602,E2 -25509.602} C_VEL
LIN {X 0,Y 138.195,Z 441.066,A -85,B 0,C 180,E1 -25514.603,E2 -25514.603} C_VEL
LIN {X 0,Y 144.538,Z 434.543,A -85,B 0,C 180,E1 -25518.911,E2 -25518.911} C_VEL
LIN {X 0,Y 150.759,Z 427.134,A -85,B 0,C 180,E1 -25522.42,E2 -25522.42} C_VEL
LIN {X 0,Y 156.326,Z 419.539,A -85,B 0,C 180,E1 -25525.132,E2 -25525.132} C_VEL
LIN {X 0,Y 162.21,Z 410.284,A -85,B 0,C 180,E1 -25527.658,E2 -25527.658} C_VEL
LIN {X 0,Y 167.912,Z 399.572,A -85,B 0,C 180,E1 -25529.85,E2 -25529.85} C_VEL
LIN {X 0,Y 172.731,Z 388.337,A -85,B 0,C 180,E1 -25531.625,E2 -25531.625} C_VEL
LIN {X 0,Y 176.614,Z 377.24,A -85,B 0,C 180,E1 -25532.918,E2 -25532.918} C_VEL
LIN {X 0,Y 180.072,Z 364.249,A -85,B 0,C 180,E1 -25533.989,E2 -25533.989} C_VEL
LIN {X 0,Y 182.382,Z 351.173,A -85,B 0,C 180,E1 -25534.721,E2 -25534.721} C_VEL
LIN {X 0,Y 184.216,Z 331.454,A -85,B 0,C 180,E1 -25535.412,E2 -25535.412} C_VEL
LIN {X 0,Y 179.984,Z 323.172,A -85,B 0,C 180,E1 -25538.526,E2 -25538.526} C_VEL
LIN {X 0,Y 175.695,Z 315.601,A -85,B 0,C 180,E1 -25542.166,E2 -25542.166} C_VEL
LIN {X 0,Y 172.411,Z 310.205,A -85,B 0,C 180,E1 -25545.466,E2 -25545.466} C_VEL
LIN {X 0,Y 169.679,Z 305.911,A -85,B 0,C 180,E1 -25548.804,E2 -25548.804} C_VEL
LIN {X 0,Y 167.365,Z 302.177,A -85,B 0,C 180,E1 -25552.403,E2 -25552.403} C_VEL
LIN {X 0,Y 166.466,Z 301.111,A -85,B 0,C 180,E1 -25554.05,E2 -25554.05} C_VEL
LIN {X 0,Y 164.568,Z 297.417,A -85,B 0,C 180,E1 -25559.46,E2 -25559.46} C_VEL
LIN {X 0,Y 164.475,Z 296.94,A -85,B 0,C 180,E1 -25560,E2 -25560} C_VEL
LIN {X 0,Y 163.907,Z 296.872,A -85,B 0,C 180,E1 -25567.39,E2 -25567.39} C_VEL
LIN {X 0,Y 164.398,Z 297.315,A -85,B 0,C 180,E1 -25570.299,E2 -25570.299} C_VEL
LIN {X 0,Y 165.805,Z 300.646,A -85,B 0,C 180,E1 -25575.047,E2 -25575.047} C_VEL
LIN {X 0,Y 167.357,Z 302.384,A -85,B 0,C 180,E1 -25578.041,E2 -25578.041} C_VEL
LIN {X 0,Y 170.173,Z 307.441,A -85,B 0,C 180,E1 -25582.379,E2 -25582.379} C_VEL
LIN {X 0,Y 172.945,Z 312.961,A -85,B 0,C 180,E1 -25585.747,E2 -25585.747} C_VEL
LIN {X 0,Y 176.132,Z 319.813,A -85,B 0,C 180,E1 -25588.997,E2 -25588.997} C_VEL
LIN {X 0,Y 179.582,Z 327.964,A -85,B 0,C 180,E1 -25592.058,E2 -25592.058} C_VEL
LIN {X 0,Y 183.396,Z 338.209,A -85,B 0,C 180,E1 -25595.087,E2 -25595.087} C_VEL
LIN {X 0,Y 183.656,Z 338.972,A -85,B 0,C 180,E1 -25595.284,E2 -25595.284} C_VEL
LIN {X 0,Y 181.569,Z 360.584,A -85,B 0,C 180,E1 -25596.013,E2 -25596.013} C_VEL
LIN {X 0,Y 179.139,Z 373.505,A -85,B 0,C 180,E1 -25596.69,E2 -25596.69} C_VEL
LIN {X 0,Y 175.797,Z 385.637,A -85,B 0,C 180,E1 -25597.622,E2 -25597.622} C_VEL
LIN {X 0,Y 171.425,Z 397.375,A -85,B 0,C 180,E1 -25598.835,E2 -25598.835} C_VEL
LIN {X 0,Y 166.203,Z 408.699,A -85,B 0,C 180,E1 -25600.435,E2 -25600.435} C_VEL
LIN {X 0,Y 160.644,Z 418.92,A -85,B 0,C 180,E1 -25602.416,E2 -25602.416} C_VEL
LIN {X 0,Y 155.237,Z 427.306,A -85,B 0,C 180,E1 -25604.516,E2 -25604.516} C_VEL
LIN {X 0,Y 148.552,Z 436.419,A -85,B 0,C 180,E1 -25607.609,E2 -25607.609} C_VEL
